LIN {X -0.037,Y -557.500,Z 807.101,A 0.000,B 0.000,C 90.000,E1 54.116} C_DIS
LIN {X -0.116,Y -555.159,Z 807.096,A 0.000,B 0.000,C 90.000,E1 53.290} C_DIS
LIN {X 0.105,Y -552.482,Z 807.091,A 0.000,B 0.000,C 90.000,E1 52.431} C_DIS
LIN {X -0.199,Y -550.629,Z 807.088,A 0.000,B 0.000,C 90.000,E1 51.904} C_DIS
LIN {X -0.029,Y -547.445,Z 807.084,A 0.000,B 0.000,C 90.000,E1 51.045} C_DIS
LIN {X -0.014,Y -545.178,Z 807.081,A 0.000,B 0.000,C 90.000,E1 50.481} C_DIS
LIN {X 0.251,Y -542.163,Z 807.077,A 0.000,B 0.000,C 90.000,E1 49.747} C_DIS
LIN {X -0.102,Y -537.935,Z 807.072,A 0.000,B 0.000,C 90.000,E1 48.933} C_DIS
LIN {X 0.083,Y -535.749,Z 807.069,A 0.000,B 0.000,C 90.000,E1 48.485} C_DIS
LIN {X -0.157,Y -531.502,Z 807.065,A 0.000,B 0.000,C 90.000,E1 47.796} C_DIS
LIN {X -0.128,Y -527.918,Z 807.062,A 0.000,B 0.000,C 90.000,E1 47.229} C_DIS
LIN {X 0.151,Y -523.761,Z 807.059,A 0.000,B 0.000,C 90.000,E1 46.620} C_DIS
LIN {X 0.098,Y -519.337,Z 807.056,A 0.000,B 0.000,C 90.000,E1 46.053} C_DIS
LIN {X 0.255,Y -514.772,Z 807.053,A 0.000,B 0.000,C 90.000,E1 45.486} C_DIS
LIN {X -0.036,Y -509.682,Z 807.050,A 0.000,B 0.000,C 90.000,E1 44.960} C_DIS
LIN {X 0.108,Y -505.640,Z 807.047,A 0.000,B 0.000,C 90.000,E1 44.514} C_DIS
LIN {X 0.235,Y -499.901,Z 807.044,A 0.000,B 0.000,C 90.000,E1 43.947} C_DIS
LIN {X -0.053,Y -495.627,Z 807.042,A 0.000,B 0.000,C 90.000,E1 43.581} C_DIS
LIN {X 0.080,Y -491.199,Z 807.040,A 0.000,B 0.000,C 90.000,E1 43.176} C_DIS
LIN {X -0.089,Y -484.986,Z 807.037,A 0.000,B 0.000,C 90.000,E1 42.690} C_DIS
LIN {X -0.041,Y -478.670,Z 807.034,A 0.000,B 0.000,C 90.000,E1 42.204} C_DIS
LIN {X 0.235,Y -470.752,Z 807.031,A 0.000,B 0.000,C 90.000,E1 41.595} C_DIS
LIN {X 0.146,Y -458.002,Z 807.026,A 0.000,B 0.000,C 90.000,E1 40.701} C_DIS
LIN {X -0.258,Y -443.553,Z 807.021,A 0.000,B 0.000,C 90.000,E1 39.725} C_DIS
LIN {X 0.027,Y -425.013,Z 807.013,A 0.000,B 0.000,C 90.000,E1 38.302} C_DIS
LIN {X 0.066,Y -412.541,Z 807.007,A 0.000,B 0.000,C 90.000,E1 37.282} C_DIS
LIN {X 0.050,Y -406.587,Z 807.004,A 0.000,B 0.000,C 90.000,E1 36.744} C_DIS
LIN {X -0.054,Y -402.832,Z 807.002,A 0.000,B 0.000,C 90.000,E1 36.377} C_DIS
LIN {X -0.143,Y -400.931,Z 807.001,A 0.000,B 0.000,C 90.000,E1 36.171} C_DIS
LIN {X 0.068,Y -400.912,Z 807.001,A 0.000,B 0.000,C 90.000,E1 36.137} C_DIS
LIN {X 0.061,Y -393.935,Z 806.977,A 0.000,B 0.000,C 90.000,E1 31.926} C_DIS
LIN {X 0.057,Y -393.844,Z 806.977,A 0.000,B 0.000,C 90.000,E1 31.750} C_DIS
LIN {X 0.223,Y -394.432,Z 806.968,A 0.000,B 0.000,C 90.000,E1 30.129} C_DIS
LIN {X -0.005,Y -395.827,Z 806.952,A 0.000,B 0.000,C 90.000,E1 27.334} C_DIS
LIN {X 0.124,Y -397.370,Z 806.938,A 0.000,B 0.000,C 90.000,E1 24.847} C_DIS
LIN {X 0.194,Y -398.558,Z 806.928,A 0.000,B 0.000,C 90.000,E1 23.078} C_DIS
LIN {X 0.069,Y -401.201,Z 806.911,A 0.000,B 0.000,C 90.000,E1 19.939} C_DIS
LIN {X 0.024,Y -404.592,Z 806.893,A 0.000,B 0.000,C 90.000,E1 16.804} C_DIS
LIN {X -0.103,Y -410.004,Z 806.872,A 0.000,B 0.000,C 90.000,E1 13.008} C_DIS
LIN {X -0.164,Y -413.482,Z 806.861,A 0.000,B 0.000,C 90.000,E1 10.950} C_DIS
LIN {X 0.106,Y -417.010,Z 806.849,A 0.000,B 0.000,C 90.000,E1 8.859} C_DIS
LIN {X -0.011,Y -420.720,Z 806.838,A 0.000,B 0.000,C 90.000,E1 6.834} C_DIS
LIN {X -0.173,Y -423.819,Z 806.829,A 0.000,B 0.000,C 90.000,E1 5.163} C_DIS
LIN {X -0.111,Y -428.905,Z 806.814,A 0.000,B 0.000,C 90.000,E1 2.465} C_DIS
LIN {X -0.089,Y -432.974,Z 806.803,A 0.000,B 0.000,C 90.000,E1 0.458} C_DIS
LIN {X 0.106,Y -437.263,Z 806.792,A 0.000,B 0.000,C 90.000,E1 358.453} C_DIS
LIN {X 0.025,Y -442.582,Z 806.779,A 0.000,B 0.000,C 90.000,E1 356.159} C_DIS
LIN {X -0.014,Y -447.421,Z 806.768,A 0.000,B 0.000,C 90.000,E1 354.204} C_DIS
LIN {X 0.034,Y -449.816,Z 806.762,A 0.000,B 0.000,C 90.000,E1 353.223} C_DIS
LIN {X -0.171,Y -454.610,Z 806.752,A 0.000,B 0.000,C 90.000,E1 351.310} C_DIS
LIN {X 0.180,Y -458.005,Z 806.745,A 0.000,B 0.000,C 90.000,E1 349.982} C_DIS
LIN {X -0.105,Y -461.068,Z 806.740,A 0.000,B 0.000,C 90.000,E1 349.218} C_DIS
LIN {X -0.029,Y -461.819,Z 806.739,A 0.000,B 0.000,C 90.000,E1 349.050} C_DIS
LIN {X -0.071,Y -464.733,Z 806.737,A 0.000,B 0.000,C 90.000,E1 348.578} C_DIS
LIN {X -0.200,Y -469.773,Z 806.734,A 0.000,B 0.000,C 90.000,E1 348.049} C_DIS
LIN {X -0.183,Y -473.009,Z 806.732,A 0.000,B 0.000,C 90.000,E1 347.757} C_DIS
LIN {X -0.111,Y -477.733,Z 806.730,A 0.000,B 0.000,C 90.000,E1 347.353} C_DIS
LIN {X 0.184,Y -498.420,Z 806.722,A 0.000,B 0.000,C 90.000,E1 345.880} C_DIS
LIN {X -0.191,Y -515.872,Z 806.715,A 0.000,B 0.000,C 90.000,E1 344.755} C_DIS
LIN {X 0.127,Y -528.321,Z 806.711,A 0.000,B 0.000,C 90.000,E1 343.866} C_DIS
LIN {X -0.178,Y -537.489,Z 806.707,A 0.000,B 0.000,C 90.000,E1 343.251} C_DIS
LIN {X 0.096,Y -544.938,Z 806.704,A 0.000,B 0.000,C 90.000,E1 342.670} C_DIS
LIN {X -0.147,Y -553.624,Z 806.700,A 0.000,B 0.000,C 90.000,E1 342.000} C_DIS
LIN {X -0.050,Y -557.840,Z 806.698,A 0.000,B 0.000,C 90.000,E1 341.638} C_DIS
LIN {X -0.131,Y -563.251,Z 806.695,A 0.000,B 0.000,C 90.000,E1 341.148} C_DIS
LIN {X 0.178,Y -568.543,Z 806.692,A 0.000,B 0.000,C 90.000,E1 340.604} C_DIS
LIN {X -0.137,Y -572.364,Z 806.690,A 0.000,B 0.000,C 90.000,E1 340.242} C_DIS
LIN {X -0.189,Y -578.188,Z 806.686,A 0.000,B 0.000,C 90.000,E1 339.571} C_DIS
LIN {X 0.115,Y -581.525,Z 806.684,A 0.000,B 0.000,C 90.000,E1 339.135} C_DIS
LIN {X 0.028,Y -587.428,Z 806.680,A 0.000,B 0.000,C 90.000,E1 338.337} C_DIS
LIN {X 0.110,Y -591.139,Z 806.677,A 0.000,B 0.000,C 90.000,E1 337.794} C_DIS
LIN {X 0.111,Y -596.462,Z 806.672,A 0.000,B 0.000,C 90.000,E1 336.997} C_DIS
LIN {X -0.149,Y -601.425,Z 806.668,A 0.000,B 0.000,C 90.000,E1 336.230} C_DIS
LIN {X -0.107,Y -607.823,Z 806.662,A 0.000,B 0.000,C 90.000,E1 335.177} C_DIS
LIN {X -0.265,Y -613.183,Z 806.657,A 0.000,B 0.000,C 90.000,E1 334.280} C_DIS
LIN {X 0.183,Y -619.697,Z 806.651,A 0.000,B 0.000,C 90.000,E1 333.076} C_DIS
LIN {X -0.384,Y -625.175,Z 806.645,A 0.000,B 0.000,C 90.000,E1 332.103} C_DIS
LIN {X -0.041,Y -629.543,Z 806.640,A 0.000,B 0.000,C 90.000,E1 331.179} C_DIS
LIN {X 0.381,Y -634.362,Z 806.634,A 0.000,B 0.000,C 90.000,E1 330.127} C_DIS
LIN {X -0.011,Y -639.079,Z 806.629,A 0.000,B 0.000,C 90.000,E1 329.154} C_DIS
LIN {X -0.081,Y -642.409,Z 806.625,A 0.000,B 0.000,C 90.000,E1 328.408} C_DIS
LIN {X -0.116,Y -645.450,Z 806.620,A 0.000,B 0.000,C 90.000,E1 327.661} C_DIS
LIN {X -0.167,Y -650.317,Z 806.613,A 0.000,B 0.000,C 90.000,E1 326.421} C_DIS
LIN {X -0.125,Y -653.040,Z 806.609,A 0.000,B 0.000,C 90.000,E1 325.674} C_DIS
LIN {X -0.141,Y -656.385,Z 806.604,A 0.000,B 0.000,C 90.000,E1 324.689} C_DIS
LIN {X -0.112,Y -659.436,Z 806.598,A 0.000,B 0.000,C 90.000,E1 323.703} C_DIS
LIN {X -0.132,Y -661.689,Z 806.594,A 0.000,B 0.000,C 90.000,E1 322.970} C_DIS
LIN {X -0.067,Y -665.082,Z 806.587,A 0.000,B 0.000,C 90.000,E1 321.743} C_DIS
LIN {X 0.043,Y -668.206,Z 806.581,A 0.000,B 0.000,C 90.000,E1 320.517} C_DIS
LIN {X 0.111,Y -670.998,Z 806.574,A 0.000,B 0.000,C 90.000,E1 319.299} C_DIS
LIN {X 0.214,Y -673.109,Z 806.569,A 0.000,B 0.000,C 90.000,E1 318.324} C_DIS
LIN {X -0.161,Y -675.018,Z 806.563,A 0.000,B 0.000,C 90.000,E1 317.391} C_DIS
LIN {X -0.450,Y -677.649,Z 806.555,A 0.000,B 0.000,C 90.000,E1 315.972} C_DIS
LIN {X -0.416,Y -678.098,Z 806.554,A 0.000,B 0.000,C 90.000,E1 315.729} C_DIS
LIN {X -0.174,Y -680.133,Z 806.546,A 0.000,B 0.000,C 90.000,E1 314.271} C_DIS
LIN {X 0.005,Y -681.446,Z 806.541,A 0.000,B 0.000,C 90.000,E1 313.299} C_DIS
LIN {X 0.284,Y -682.974,Z 806.534,A 0.000,B 0.000,C 90.000,E1 312.081} C_DIS
LIN {X 0.081,Y -684.417,Z 806.527,A 0.000,B 0.000,C 90.000,E1 310.906} C_DIS
LIN {X 0.018,Y -685.924,Z 806.519,A 0.000,B 0.000,C 90.000,E1 309.483} C_DIS
LIN {X -0.072,Y -687.086,Z 806.513,A 0.000,B 0.000,C 90.000,E1 308.302} C_DIS
LIN {X 0.024,Y -688.401,Z 806.505,A 0.000,B 0.000,C 90.000,E1 306.870} C_DIS
LIN {X 0.147,Y -689.583,Z 806.497,A 0.000,B 0.000,C 90.000,E1 305.438} C_DIS
LIN {X -0.142,Y -690.502,Z 806.490,A 0.000,B 0.000,C 90.000,E1 304.278} C_DIS
LIN {X -0.163,Y -691.695,Z 806.481,A 0.000,B 0.000,C 90.000,E1 302.625} C_DIS
LIN {X 0.056,Y -693.170,Z 806.471,A 0.000,B 0.000,C 90.000,E1 300.718} C_DIS
LIN {X -0.296,Y -694.103,Z 806.463,A 0.000,B 0.000,C 90.000,E1 299.333} C_DIS
LIN {X 0.228,Y -695.151,Z 806.454,A 0.000,B 0.000,C 90.000,E1 297.641} C_DIS
LIN {X -0.215,Y -696.425,Z 806.443,A 0.000,B 0.000,C 90.000,E1 295.796} C_DIS
LIN {X -0.104,Y -697.186,Z 806.438,A 0.000,B 0.000,C 90.000,E1 294.847} C_DIS
LIN {X -0.219,Y -697.383,Z 806.435,A 0.000,B 0.000,C 90.000,E1 294.387} C_DIS
LIN {X 0.039,Y -697.356,Z 806.434,A 0.000,B 0.000,C 90.000,E1 294.131} C_DIS
LIN {X 0.273,Y -696.938,Z 806.432,A 0.000,B 0.000,C 90.000,E1 293.643} C_DIS
LIN {X -0.110,Y -696.321,Z 806.430,A 0.000,B 0.000,C 90.000,E1 293.439} C_DIS
LIN {X 0.121,Y -694.445,Z 806.428,A 0.000,B 0.000,C 90.000,E1 292.950} C_DIS
LIN {X 0.245,Y -693.752,Z 806.427,A 0.000,B 0.000,C 90.000,E1 292.823} C_DIS
LIN {X 0.100,Y -692.715,Z 806.426,A 0.000,B 0.000,C 90.000,E1 292.717} C_DIS
LIN {X 0.220,Y -691.283,Z 806.426,A 0.000,B 0.000,C 90.000,E1 292.589} C_DIS
LIN {X 0.129,Y -686.698,Z 806.424,A 0.000,B 0.000,C 90.000,E1 292.280} C_DIS
LIN {X -0.136,Y -685.084,Z 806.423,A 0.000,B 0.000,C 90.000,E1 292.206} C_DIS
LIN {X 0.232,Y -682.669,Z 806.423,A 0.000,B 0.000,C 90.000,E1 292.078} C_DIS
LIN {X 0.207,Y -675.226,Z 806.422,A 0.000,B 0.000,C 90.000,E1 291.844} C_DIS
LIN {X 0.189,Y -673.325,Z 806.421,A 0.000,B 0.000,C 90.000,E1 291.791} C_DIS
LIN {X -0.184,Y -664.792,Z 806.420,A 0.000,B 0.000,C 90.000,E1 291.663} C_DIS
LIN {X -0.168,Y -648.502,Z 806.419,A 0.000,B 0.000,C 90.000,E1 291.408} C_DIS
LIN {X 0.368,Y -627.611,Z 806.417,A 0.000,B 0.000,C 90.000,E1 290.972} C_DIS
LIN {X -0.380,Y -614.207,Z 806.415,A 0.000,B 0.000,C 90.000,E1 290.737} C_DIS
LIN {X 0.116,Y -604.662,Z 806.414,A 0.000,B 0.000,C 90.000,E1 290.429} C_DIS
LIN {X -0.075,Y -595.597,Z 806.412,A 0.000,B 0.000,C 90.000,E1 290.120} C_DIS
LIN {X -0.078,Y -590.879,Z 806.411,A 0.000,B 0.000,C 90.000,E1 289.939} C_DIS
LIN {X -0.260,Y -587.841,Z 806.410,A 0.000,B 0.000,C 90.000,E1 289.812} C_DIS
LIN {X 0.019,Y -585.447,Z 806.409,A 0.000,B 0.000,C 90.000,E1 289.631} C_DIS
LIN {X -0.206,Y -582.531,Z 806.408,A 0.000,B 0.000,C 90.000,E1 289.504} C_DIS
LIN {X 0.311,Y -582.496,Z 806.408,A 0.000,B 0.000,C 90.000,E1 289.450} C_DIS
LIN {X 0.310,Y -581.681,Z 806.407,A 0.000,B 0.000,C 90.000,E1 289.268} C_DIS
LIN {X -0.111,Y -582.551,Z 806.405,A 0.000,B 0.000,C 90.000,E1 288.906} C_DIS
LIN {X 0.284,Y -583.583,Z 806.404,A 0.000,B 0.000,C 90.000,E1 288.598} C_DIS
LIN {X 0.140,Y -587.254,Z 806.400,A 0.000,B 0.000,C 90.000,E1 287.946} C_DIS
LIN {X 0.160,Y -591.295,Z 806.396,A 0.000,B 0.000,C 90.000,E1 287.275} C_DIS
LIN {X -0.028,Y -595.685,Z 806.392,A 0.000,B 0.000,C 90.000,E1 286.496} C_DIS
LIN {X 0.245,Y -596.903,Z 806.390,A 0.000,B 0.000,C 90.000,E1 286.205} C_DIS
LIN {X 0.109,Y -600.031,Z 806.386,A 0.000,B 0.000,C 90.000,E1 285.426} C_DIS
LIN {X -0.178,Y -600.898,Z 806.384,A 0.000,B 0.000,C 90.000,E1 285.190} C_DIS
LIN {X -0.006,Y -602.048,Z 806.381,A 0.000,B 0.000,C 90.000,E1 284.647} C_DIS
LIN {X 0.022,Y -602.938,Z 806.378,A 0.000,B 0.000,C 90.000,E1 284.120} C_DIS
LIN {X -0.254,Y -603.285,Z 806.377,A 0.000,B 0.000,C 90.000,E1 283.883} C_DIS
LIN {X -0.214,Y -603.288,Z 806.374,A 0.000,B 0.000,C 90.000,E1 283.355} C_DIS
LIN {X -0.171,Y -602.957,Z 806.371,A 0.000,B 0.000,C 90.000,E1 282.827} C_DIS
LIN {X 0.144,Y -602.625,Z 806.370,A 0.000,B 0.000,C 90.000,E1 282.535} C_DIS
LIN {X 0.184,Y -601.388,Z 806.367,A 0.000,B 0.000,C 90.000,E1 282.007} C_DIS
LIN {X 0.215,Y -599.980,Z 806.364,A 0.000,B 0.000,C 90.000,E1 281.478} C_DIS
LIN {X 0.235,Y -597.951,Z 806.361,A 0.000,B 0.000,C 90.000,E1 280.950} C_DIS
LIN {X -0.256,Y -596.181,Z 806.359,A 0.000,B 0.000,C 90.000,E1 280.602} C_DIS
LIN {X 0.035,Y -594.900,Z 806.357,A 0.000,B 0.000,C 90.000,E1 280.310} C_DIS
LIN {X -0.088,Y -591.719,Z 806.354,A 0.000,B 0.000,C 90.000,E1 279.792} C_DIS
LIN {X 0.077,Y -588.827,Z 806.352,A 0.000,B 0.000,C 90.000,E1 279.378} C_DIS
LIN {X 0.242,Y -586.579,Z 806.351,A 0.000,B 0.000,C 90.000,E1 279.095} C_DIS
LIN {X 0.126,Y -585.159,Z 806.350,A 0.000,B 0.000,C 90.000,E1 278.973} C_DIS
LIN {X -0.083,Y -583.486,Z 806.349,A 0.000,B 0.000,C 90.000,E1 278.859} C_DIS
LIN {X -0.093,Y -581.758,Z 806.349,A 0.000,B 0.000,C 90.000,E1 278.746} C_DIS
LIN {X 0.246,Y -577.851,Z 806.347,A 0.000,B 0.000,C 90.000,E1 278.511} C_DIS
LIN {X -0.045,Y -569.845,Z 806.346,A 0.000,B 0.000,C 90.000,E1 278.276} C_DIS
LIN {X 0.054,Y -559.795,Z 806.345,A 0.000,B 0.000,C 90.000,E1 278.049} C_DIS
LIN {X 0.236,Y -556.972,Z 806.345,A 0.000,B 0.000,C 90.000,E1 277.992} C_DIS
LIN {X -0.197,Y -553.699,Z 806.344,A 0.000,B 0.000,C 90.000,E1 277.936} C_DIS
LIN {X 0.061,Y -553.337,Z 806.344,A 0.000,B 0.000,C 90.000,E1 277.871} C_DIS
LIN {X -0.192,Y -552.403,Z 806.343,A 0.000,B 0.000,C 90.000,E1 277.757} C_DIS
LIN {X -0.274,Y -551.492,Z 806.342,A 0.000,B 0.000,C 90.000,E1 277.644} C_DIS
LIN {X 0.188,Y -551.453,Z 806.342,A 0.000,B 0.000,C 90.000,E1 277.587} C_DIS
LIN {X 0.146,Y -551.448,Z 806.342,A 0.000,B 0.000,C 90.000,E1 277.587} C_DIS
LIN {X -0.026,Y -551.293,Z 806.341,A 0.000,B 0.000,C 90.000,E1 277.409} C_DIS
LIN {X -0.227,Y -550.912,Z 806.340,A 0.000,B 0.000,C 90.000,E1 277.239} C_DIS
LIN {X 0.166,Y -549.933,Z 806.332,A 0.000,B 0.000,C 90.000,E1 275.796} C_DIS
LIN {X -0.107,Y -549.514,Z 806.326,A 0.000,B 0.000,C 90.000,E1 274.702} C_DIS
LIN {X 0.119,Y -548.833,Z 806.320,A 0.000,B 0.000,C 90.000,E1 273.555} C_DIS
LIN {X -0.208,Y -548.137,Z 806.314,A 0.000,B 0.000,C 90.000,E1 272.465} C_DIS
LIN {X 0.135,Y -546.720,Z 806.303,A 0.000,B 0.000,C 90.000,E1 270.458} C_DIS
LIN {X -0.195,Y -545.795,Z 806.295,A 0.000,B 0.000,C 90.000,E1 269.083} C_DIS
LIN {X 0.144,Y -544.235,Z 806.282,A 0.000,B 0.000,C 90.000,E1 266.788} C_DIS
LIN {X -0.129,Y -543.053,Z 806.271,A 0.000,B 0.000,C 90.000,E1 264.837} C_DIS
LIN {X 0.119,Y -542.072,Z 806.263,A 0.000,B 0.000,C 90.000,E1 263.394} C_DIS
LIN {X -0.186,Y -540.898,Z 806.256,A 0.000,B 0.000,C 90.000,E1 262.008} C_DIS
LIN {X 0.082,Y -539.379,Z 806.246,A 0.000,B 0.000,C 90.000,E1 260.274} C_DIS
LIN {X -0.171,Y -538.251,Z 806.240,A 0.000,B 0.000,C 90.000,E1 259.162} C_DIS
LIN {X 0.158,Y -536.897,Z 806.232,A 0.000,B 0.000,C 90.000,E1 257.701} C_DIS
LIN {X 0.110,Y -535.129,Z 806.222,A 0.000,B 0.000,C 90.000,E1 255.992} C_DIS
LIN {X 0.201,Y -532.815,Z 806.211,A 0.000,B 0.000,C 90.000,E1 253.976} C_DIS
LIN {X -0.320,Y -530.792,Z 806.202,A 0.000,B 0.000,C 90.000,E1 252.308} C_DIS
LIN {X -0.240,Y -529.077,Z 806.194,A 0.000,B 0.000,C 90.000,E1 250.859} C_DIS
LIN {X -0.194,Y -527.535,Z 806.187,A 0.000,B 0.000,C 90.000,E1 249.699} C_DIS
LIN {X 0.002,Y -525.491,Z 806.179,A 0.000,B 0.000,C 90.000,E1 248.230} C_DIS
LIN {X -0.132,Y -523.365,Z 806.171,A 0.000,B 0.000,C 90.000,E1 246.794} C_DIS
LIN {X -0.300,Y -521.192,Z 806.163,A 0.000,B 0.000,C 90.000,E1 245.357} C_DIS
LIN {X 0.037,Y -519.355,Z 806.156,A 0.000,B 0.000,C 90.000,E1 244.152} C_DIS
LIN {X 0.027,Y -515.813,Z 806.145,A 0.000,B 0.000,C 90.000,E1 242.103} C_DIS
LIN {X -0.291,Y -513.076,Z 806.137,A 0.000,B 0.000,C 90.000,E1 240.667} C_DIS
LIN {X 0.035,Y -510.317,Z 806.129,A 0.000,B 0.000,C 90.000,E1 239.154} C_DIS
LIN {X -0.195,Y -507.992,Z 806.122,A 0.000,B 0.000,C 90.000,E1 237.995} C_DIS
LIN {X -0.135,Y -504.791,Z 806.114,A 0.000,B 0.000,C 90.000,E1 236.501} C_DIS
LIN {X -0.158,Y -502.316,Z 806.107,A 0.000,B 0.000,C 90.000,E1 235.308} C_DIS
LIN {X -0.213,Y -499.557,Z 806.101,A 0.000,B 0.000,C 90.000,E1 234.116} C_DIS
LIN {X 0.114,Y -495.036,Z 806.091,A 0.000,B 0.000,C 90.000,E1 232.271} C_DIS
LIN {X -0.002,Y -492.789,Z 806.085,A 0.000,B 0.000,C 90.000,E1 231.376} C_DIS
LIN {X 0.031,Y -485.624,Z 806.069,A 0.000,B 0.000,C 90.000,E1 228.324} C_DIS
LIN {X -0.212,Y -480.238,Z 806.055,A 0.000,B 0.000,C 90.000,E1 225.891} C_DIS
LIN {X -0.167,Y -476.113,Z 806.045,A 0.000,B 0.000,C 90.000,E1 224.028} C_DIS
LIN {X 0.026,Y -472.717,Z 806.036,A 0.000,B 0.000,C 90.000,E1 222.447} C_DIS
LIN {X 0.097,Y -467.428,Z 806.022,A 0.000,B 0.000,C 90.000,E1 219.930} C_DIS
LIN {X -0.144,Y -464.126,Z 806.013,A 0.000,B 0.000,C 90.000,E1 218.382} C_DIS
LIN {X -0.084,Y -460.861,Z 806.004,A 0.000,B 0.000,C 90.000,E1 216.790} C_DIS
LIN {X 0.220,Y -455.527,Z 805.990,A 0.000,B 0.000,C 90.000,E1 214.199} C_DIS
LIN {X -0.038,Y -452.264,Z 805.981,A 0.000,B 0.000,C 90.000,E1 212.625} C_DIS
LIN {X 0.106,Y -448.344,Z 805.971,A 0.000,B 0.000,C 90.000,E1 210.669} C_DIS
LIN {X -0.078,Y -444.464,Z 805.960,A 0.000,B 0.000,C 90.000,E1 208.743} C_DIS
LIN {X -0.224,Y -441.287,Z 805.951,A 0.000,B 0.000,C 90.000,E1 207.129} C_DIS
LIN {X -0.202,Y -437.595,Z 805.940,A 0.000,B 0.000,C 90.000,E1 205.155} C_DIS
LIN {X 0.121,Y -434.327,Z 805.930,A 0.000,B 0.000,C 90.000,E1 203.462} C_DIS
LIN {X -0.003,Y -429.806,Z 805.918,A 0.000,B 0.000,C 90.000,E1 201.153} C_DIS
LIN {X -0.114,Y -424.685,Z 805.903,A 0.000,B 0.000,C 90.000,E1 198.489} C_DIS
LIN {X 0.070,Y -420.794,Z 805.891,A 0.000,B 0.000,C 90.000,E1 196.441} C_DIS
LIN {X -0.126,Y -417.498,Z 805.882,A 0.000,B 0.000,C 90.000,E1 194.773} C_DIS
LIN {X -0.090,Y -414.261,Z 805.873,A 0.000,B 0.000,C 90.000,E1 193.063} C_DIS
LIN {X -0.093,Y -410.442,Z 805.861,A 0.000,B 0.000,C 90.000,E1 191.007} C_DIS
LIN {X 0.055,Y -406.743,Z 805.850,A 0.000,B 0.000,C 90.000,E1 188.916} C_DIS
LIN {X 0.052,Y -403.462,Z 805.840,A 0.000,B 0.000,C 90.000,E1 187.182} C_DIS
LIN {X -0.008,Y -400.980,Z 805.832,A 0.000,B 0.000,C 90.000,E1 185.796} C_DIS
LIN {X -0.177,Y -397.974,Z 805.823,A 0.000,B 0.000,C 90.000,E1 184.069} C_DIS
LIN {X -0.063,Y -392.546,Z 805.801,A 0.000,B 0.000,C 90.000,E1 180.172} C_DIS
LIN {X 0.175,Y -389.636,Z 805.787,A 0.000,B 0.000,C 90.000,E1 177.650} C_DIS
LIN {X -0.073,Y -388.507,Z 805.781,A 0.000,B 0.000,C 90.000,E1 176.617} C_DIS
LIN {X 0.081,Y -385.777,Z 805.767,A 0.000,B 0.000,C 90.000,E1 174.090} C_DIS
LIN {X -0.030,Y -383.509,Z 805.755,A 0.000,B 0.000,C 90.000,E1 171.951} C_DIS
LIN {X -0.048,Y -381.888,Z 805.745,A 0.000,B 0.000,C 90.000,E1 170.151} C_DIS
LIN {X 0.141,Y -379.406,Z 805.729,A 0.000,B 0.000,C 90.000,E1 167.229} C_DIS
LIN {X 0.054,Y -377.533,Z 805.715,A 0.000,B 0.000,C 90.000,E1 164.700} C_DIS
LIN {X -0.181,Y -375.922,Z 805.697,A 0.000,B 0.000,C 90.000,E1 161.456} C_DIS
LIN {X -0.183,Y -375.346,Z 805.683,A 0.000,B 0.000,C 90.000,E1 158.901} C_DIS
LIN {X -0.185,Y -375.706,Z 805.664,A 0.000,B 0.000,C 90.000,E1 155.613} C_DIS
LIN {X 0.074,Y -376.792,Z 805.652,A 0.000,B 0.000,C 90.000,E1 153.384} C_DIS
LIN {X 0.011,Y -379.478,Z 805.638,A 0.000,B 0.000,C 90.000,E1 150.845} C_DIS
LIN {X -0.087,Y -382.025,Z 805.630,A 0.000,B 0.000,C 90.000,E1 149.410} C_DIS
LIN {X 0.074,Y -383.792,Z 805.626,A 0.000,B 0.000,C 90.000,E1 148.663} C_DIS
LIN {X -0.099,Y -386.398,Z 805.621,A 0.000,B 0.000,C 90.000,E1 147.788} C_DIS
LIN {X -0.084,Y -388.278,Z 805.618,A 0.000,B 0.000,C 90.000,E1 147.248} C_DIS
LIN {X -0.097,Y -390.773,Z 805.614,A 0.000,B 0.000,C 90.000,E1 146.548} C_DIS
LIN {X 0.143,Y -393.979,Z 805.610,A 0.000,B 0.000,C 90.000,E1 145.801} C_DIS
LIN {X -0.041,Y -396.643,Z 805.607,A 0.000,B 0.000,C 90.000,E1 145.308} C_DIS
LIN {X -0.078,Y -400.780,Z 805.603,A 0.000,B 0.000,C 90.000,E1 144.609} C_DIS
LIN {X 0.020,Y -404.295,Z 805.600,A 0.000,B 0.000,C 90.000,E1 144.069} C_DIS
LIN {X -0.214,Y -413.312,Z 805.594,A 0.000,B 0.000,C 90.000,E1 142.924} C_DIS
LIN {X 0.000,Y -424.271,Z 805.587,A 0.000,B 0.000,C 90.000,E1 141.662} C_DIS
LIN {X 0.031,Y -429.654,Z 805.583,A 0.000,B 0.000,C 90.000,E1 141.009} C_DIS
LIN {X -0.130,Y -439.865,Z 805.576,A 0.000,B 0.000,C 90.000,E1 139.703} C_DIS
LIN {X 0.104,Y -446.170,Z 805.572,A 0.000,B 0.000,C 90.000,E1 138.852} C_DIS
LIN {X 0.152,Y -455.314,Z 805.565,A 0.000,B 0.000,C 90.000,E1 137.715} C_DIS
LIN {X 0.218,Y -460.035,Z 805.562,A 0.000,B 0.000,C 90.000,E1 137.067} C_DIS
LIN {X -0.014,Y -464.335,Z 805.558,A 0.000,B 0.000,C 90.000,E1 136.458} C_DIS
LIN {X -0.172,Y -477.324,Z 805.547,A 0.000,B 0.000,C 90.000,E1 134.433} C_DIS
LIN {X 0.176,Y -483.191,Z 805.542,A 0.000,B 0.000,C 90.000,E1 133.461} C_DIS
LIN {X 0.167,Y -491.525,Z 805.534,A 0.000,B 0.000,C 90.000,E1 132.081} C_DIS
LIN {X -0.196,Y -494.989,Z 805.531,A 0.000,B 0.000,C 90.000,E1 131.515} C_DIS
LIN {X -0.143,Y -504.022,Z 805.521,A 0.000,B 0.000,C 90.000,E1 129.850} C_DIS
LIN {X 0.058,Y -511.764,Z 805.513,A 0.000,B 0.000,C 90.000,E1 128.338} C_DIS
LIN {X 0.002,Y -518.944,Z 805.505,A 0.000,B 0.000,C 90.000,E1 126.870} C_DIS
LIN {X -0.208,Y -524.279,Z 805.498,A 0.000,B 0.000,C 90.000,E1 125.724} C_DIS
LIN {X 0.107,Y -527.837,Z 805.494,A 0.000,B 0.000,C 90.000,E1 124.818} C_DIS
LIN {X -0.134,Y -531.610,Z 805.488,A 0.000,B 0.000,C 90.000,E1 123.833} C_DIS
LIN {X 0.122,Y -534.492,Z 805.484,A 0.000,B 0.000,C 90.000,E1 123.086} C_DIS
LIN {X -0.025,Y -538.937,Z 805.478,A 0.000,B 0.000,C 90.000,E1 121.957} C_DIS
LIN {X -0.295,Y -542.012,Z 805.473,A 0.000,B 0.000,C 90.000,E1 121.131} C_DIS
LIN {X -0.074,Y -544.846,Z 805.468,A 0.000,B 0.000,C 90.000,E1 120.256} C_DIS
LIN {X -0.075,Y -548.311,Z 805.462,A 0.000,B 0.000,C 90.000,E1 119.127} C_DIS
LIN {X 0.191,Y -551.559,Z 805.456,A 0.000,B 0.000,C 90.000,E1 117.975} C_DIS
LIN {X 0.248,Y -553.701,Z 805.451,A 0.000,B 0.000,C 90.000,E1 117.129} C_DIS
LIN {X 0.076,Y -555.541,Z 805.446,A 0.000,B 0.000,C 90.000,E1 116.309} C_DIS
LIN {X 0.247,Y -557.849,Z 805.439,A 0.000,B 0.000,C 90.000,E1 114.899} C_DIS
LIN {X -0.089,Y -559.312,Z 805.432,A 0.000,B 0.000,C 90.000,E1 113.823} C_DIS
LIN {X 0.103,Y -560.602,Z 805.426,A 0.000,B 0.000,C 90.000,E1 112.695} C_DIS
LIN {X -0.113,Y -561.993,Z 805.419,A 0.000,B 0.000,C 90.000,E1 111.334} C_DIS
LIN {X 0.108,Y -562.648,Z 805.414,A 0.000,B 0.000,C 90.000,E1 110.482} C_DIS
LIN {X -0.061,Y -563.241,Z 805.408,A 0.000,B 0.000,C 90.000,E1 109.396} C_DIS
LIN {X -0.037,Y -563.706,Z 805.402,A 0.000,B 0.000,C 90.000,E1 108.290} C_DIS
LIN {X 0.028,Y -564.544,Z 805.389,A 0.000,B 0.000,C 90.000,E1 106.079} C_DIS
LIN {X -0.194,Y -565.506,Z 805.379,A 0.000,B 0.000,C 90.000,E1 104.175} C_DIS
LIN {X 0.063,Y -566.969,Z 805.366,A 0.000,B 0.000,C 90.000,E1 101.951} C_DIS
LIN {X 0.186,Y -568.338,Z 805.356,A 0.000,B 0.000,C 90.000,E1 100.018} C_DIS
LIN {X -0.135,Y -569.364,Z 805.348,A 0.000,B 0.000,C 90.000,E1 98.681} C_DIS
LIN {X 0.041,Y -570.288,Z 805.341,A 0.000,B 0.000,C 90.000,E1 97.296} C_DIS
LIN {X -0.059,Y -570.807,Z 805.336,A 0.000,B 0.000,C 90.000,E1 96.486} C_DIS
LIN {X 0.084,Y -571.578,Z 805.328,A 0.000,B 0.000,C 90.000,E1 95.106} C_DIS
LIN {X 0.244,Y -572.276,Z 805.321,A 0.000,B 0.000,C 90.000,E1 93.726} C_DIS
LIN {X -0.193,Y -572.877,Z 805.313,A 0.000,B 0.000,C 90.000,E1 92.407} C_DIS
LIN {X 0.238,Y -573.574,Z 805.303,A 0.000,B 0.000,C 90.000,E1 90.458} C_DIS
LIN {X -0.046,Y -574.120,Z 805.294,A 0.000,B 0.000,C 90.000,E1 88.854} C_DIS
LIN {X 0.121,Y -574.471,Z 805.286,A 0.000,B 0.000,C 90.000,E1 87.478} C_DIS
LIN {X -0.100,Y -574.846,Z 805.277,A 0.000,B 0.000,C 90.000,E1 85.869} C_DIS
LIN {X 0.123,Y -575.129,Z 805.270,A 0.000,B 0.000,C 90.000,E1 84.489} C_DIS
LIN {X -0.230,Y -575.430,Z 805.262,A 0.000,B 0.000,C 90.000,E1 83.166} C_DIS
LIN {X 0.012,Y -575.886,Z 805.250,A 0.000,B 0.000,C 90.000,E1 80.971} C_DIS
LIN {X 0.237,Y -576.269,Z 805.239,A 0.000,B 0.000,C 90.000,E1 79.050} C_DIS
LIN {X -0.048,Y -576.392,Z 805.233,A 0.000,B 0.000,C 90.000,E1 77.993} C_DIS
LIN {X -0.118,Y -576.462,Z 805.226,A 0.000,B 0.000,C 90.000,E1 76.645} C_DIS
LIN {X 0.296,Y -576.416,Z 805.220,A 0.000,B 0.000,C 90.000,E1 75.519} C_DIS
LIN {X 0.157,Y -576.335,Z 805.214,A 0.000,B 0.000,C 90.000,E1 74.448} C_DIS
LIN {X 0.028,Y -576.153,Z 805.205,A 0.000,B 0.000,C 90.000,E1 72.834} C_DIS
LIN {X 0.245,Y -575.914,Z 805.197,A 0.000,B 0.000,C 90.000,E1 71.456} C_DIS
LIN {X 0.098,Y -575.343,Z 805.187,A 0.000,B 0.000,C 90.000,E1 69.571} C_DIS
LIN {X -0.071,Y -574.833,Z 805.179,A 0.000,B 0.000,C 90.000,E1 68.230} C_DIS
LIN {X -0.042,Y -574.206,Z 805.172,A 0.000,B 0.000,C 90.000,E1 66.869} C_DIS
LIN {X 0.203,Y -573.509,Z 805.164,A 0.000,B 0.000,C 90.000,E1 65.485} C_DIS
LIN {X 0.079,Y -572.827,Z 805.158,A 0.000,B 0.000,C 90.000,E1 64.409} C_DIS
LIN {X 0.038,Y -571.903,Z 805.150,A 0.000,B 0.000,C 90.000,E1 63.050} C_DIS
LIN {X -0.114,Y -570.918,Z 805.144,A 0.000,B 0.000,C 90.000,E1 61.975} C_DIS
LIN {X -0.022,Y -569.723,Z 805.138,A 0.000,B 0.000,C 90.000,E1 60.873} C_DIS
LIN {X 0.015,Y -568.721,Z 805.134,A 0.000,B 0.000,C 90.000,E1 60.049} C_DIS
LIN {X 0.070,Y -567.182,Z 805.128,A 0.000,B 0.000,C 90.000,E1 58.948} C_DIS
LIN {X -0.098,Y -565.423,Z 805.121,A 0.000,B 0.000,C 90.000,E1 57.867} C_DIS
LIN {X 0.016,Y -563.361,Z 805.115,A 0.000,B 0.000,C 90.000,E1 56.755} C_DIS
LIN {X 0.011,Y -561.681,Z 805.111,A 0.000,B 0.000,C 90.000,E1 55.928} C_DIS
LIN {X 0.080,Y -559.052,Z 805.105,A 0.000,B 0.000,C 90.000,E1 54.815} C_DIS
LIN {X 0.022,Y -556.875,Z 805.100,A 0.000,B 0.000,C 90.000,E1 53.989} C_DIS
LIN {X 0.186,Y -555.340,Z 805.097,A 0.000,B 0.000,C 90.000,E1 53.417} C_DIS
LIN {X -0.028,Y -552.676,Z 805.092,A 0.000,B 0.000,C 90.000,E1 52.603} C_DIS
LIN {X 0.171,Y -549.737,Z 805.088,A 0.000,B 0.000,C 90.000,E1 51.743} C_DIS
LIN {X 0.282,Y -547.660,Z 805.084,A 0.000,B 0.000,C 90.000,E1 51.170} C_DIS
LIN {X 0.028,Y -542.876,Z 805.078,A 0.000,B 0.000,C 90.000,E1 50.070} C_DIS
LIN {X -0.168,Y -540.954,Z 805.076,A 0.000,B 0.000,C 90.000,E1 49.666} C_DIS
LIN {X 0.050,Y -537.382,Z 805.072,A 0.000,B 0.000,C 90.000,E1 48.933} C_DIS
LIN {X -0.171,Y -535.154,Z 805.070,A 0.000,B 0.000,C 90.000,E1 48.528} C_DIS
LIN {X -0.016,Y -530.818,Z 805.066,A 0.000,B 0.000,C 90.000,E1 47.796} C_DIS
LIN {X 0.002,Y -527.118,Z 805.062,A 0.000,B 0.000,C 90.000,E1 47.229} C_DIS
LIN {X -0.096,Y -522.899,Z 805.059,A 0.000,B 0.000,C 90.000,E1 46.662} C_DIS
LIN {X 0.033,Y -519.564,Z 805.057,A 0.000,B 0.000,C 90.000,E1 46.215} C_DIS
LIN {X 0.055,Y -514.861,Z 805.054,A 0.000,B 0.000,C 90.000,E1 45.648} C_DIS
LIN {X 0.108,Y -509.726,Z 805.051,A 0.000,B 0.000,C 90.000,E1 45.081} C_DIS
LIN {X -0.015,Y -505.735,Z 805.048,A 0.000,B 0.000,C 90.000,E1 44.676} C_DIS
LIN {X 0.233,Y -500.133,Z 805.045,A 0.000,B 0.000,C 90.000,E1 44.109} C_DIS
LIN {X -0.004,Y -493.097,Z 805.042,A 0.000,B 0.000,C 90.000,E1 43.500} C_DIS
LIN {X 0.132,Y -488.456,Z 805.040,A 0.000,B 0.000,C 90.000,E1 43.095} C_DIS
LIN {X 0.179,Y -482.401,Z 805.037,A 0.000,B 0.000,C 90.000,E1 42.609} C_DIS
LIN {X 0.029,Y -474.527,Z 805.034,A 0.000,B 0.000,C 90.000,E1 42.043} C_DIS
LIN {X 0.207,Y -463.356,Z 805.029,A 0.000,B 0.000,C 90.000,E1 41.229} C_DIS
LIN {X -0.012,Y -445.813,Z 805.022,A 0.000,B 0.000,C 90.000,E1 40.011} C_DIS
LIN {X -0.133,Y -426.715,Z 805.015,A 0.000,B 0.000,C 90.000,E1 38.624} C_DIS
LIN {X -0.183,Y -411.107,Z 805.008,A 0.000,B 0.000,C 90.000,E1 37.363} C_DIS
LIN {X -0.135,Y -406.610,Z 805.005,A 0.000,B 0.000,C 90.000,E1 36.950} C_DIS
LIN {X -0.009,Y -401.370,Z 805.002,A 0.000,B 0.000,C 90.000,E1 36.377} C_DIS
LIN {X -0.042,Y -401.353,Z 805.002,A 0.000,B 0.000,C 90.000,E1 36.377} C_DIS
LIN {X -0.047,Y -394.198,Z 804.979,A 0.000,B 0.000,C 90.000,E1 32.133} C_DIS
LIN {X 0.157,Y -394.028,Z 804.978,A 0.000,B 0.000,C 90.000,E1 31.926} C_DIS
LIN {X 0.155,Y -394.612,Z 804.969,A 0.000,B 0.000,C 90.000,E1 30.335} C_DIS
LIN {X -0.095,Y -395.791,Z 804.955,A 0.000,B 0.000,C 90.000,E1 27.897} C_DIS
LIN {X 0.023,Y -397.253,Z 804.941,A 0.000,B 0.000,C 90.000,E1 25.412} C_DIS
LIN {X 0.091,Y -398.440,Z 804.931,A 0.000,B 0.000,C 90.000,E1 23.643} C_DIS
LIN {X 0.192,Y -401.262,Z 804.912,A 0.000,B 0.000,C 90.000,E1 20.120} C_DIS
LIN {X 0.149,Y -404.622,Z 804.895,A 0.000,B 0.000,C 90.000,E1 16.985} C_DIS
LIN {X 0.010,Y -409.449,Z 804.875,A 0.000,B 0.000,C 90.000,E1 13.536} C_DIS
LIN {X -0.026,Y -413.396,Z 804.862,A 0.000,B 0.000,C 90.000,E1 11.130} C_DIS
LIN {X -0.161,Y -416.959,Z 804.850,A 0.000,B 0.000,C 90.000,E1 9.095} C_DIS
LIN {X 0.142,Y -420.641,Z 804.839,A 0.000,B 0.000,C 90.000,E1 7.011} C_DIS
LIN {X 0.027,Y -423.765,Z 804.830,A 0.000,B 0.000,C 90.000,E1 5.334} C_DIS
LIN {X 0.149,Y -429.463,Z 804.813,A 0.000,B 0.000,C 90.000,E1 2.293} C_DIS
LIN {X 0.165,Y -434.636,Z 804.799,A 0.000,B 0.000,C 90.000,E1 359.771} C_DIS
LIN {X 0.109,Y -440.484,Z 804.784,A 0.000,B 0.000,C 90.000,E1 357.135} C_DIS
LIN {X 0.149,Y -446.026,Z 804.771,A 0.000,B 0.000,C 90.000,E1 354.837} C_DIS
LIN {X 0.053,Y -450.039,Z 804.762,A 0.000,B 0.000,C 90.000,E1 353.223} C_DIS
LIN {X -0.147,Y -454.780,Z 804.752,A 0.000,B 0.000,C 90.000,E1 351.310} C_DIS
LIN {X 0.205,Y -458.138,Z 804.745,A 0.000,B 0.000,C 90.000,E1 349.982} C_DIS
LIN {X -0.061,Y -460.848,Z 804.740,A 0.000,B 0.000,C 90.000,E1 349.218} C_DIS
LIN {X -0.199,Y -463.187,Z 804.737,A 0.000,B 0.000,C 90.000,E1 348.757} C_DIS
LIN {X 0.089,Y -465.609,Z 804.735,A 0.000,B 0.000,C 90.000,E1 348.342} C_DIS
LIN {X 0.069,Y -469.780,Z 804.733,A 0.000,B 0.000,C 90.000,E1 347.881} C_DIS
LIN {X 0.205,Y -473.528,Z 804.731,A 0.000,B 0.000,C 90.000,E1 347.521} C_DIS
LIN {X -0.123,Y -479.550,Z 804.728,A 0.000,B 0.000,C 90.000,E1 347.061} C_DIS
LIN {X -0.198,Y -503.485,Z 804.719,A 0.000,B 0.000,C 90.000,E1 345.408} C_DIS
LIN {X -0.146,Y -517.729,Z 804.714,A 0.000,B 0.000,C 90.000,E1 344.448} C_DIS
LIN {X 0.046,Y -528.645,Z 804.709,A 0.000,B 0.000,C 90.000,E1 343.685} C_DIS
LIN {X 0.110,Y -537.759,Z 804.706,A 0.000,B 0.000,C 90.000,E1 343.032} C_DIS
LIN {X -0.038,Y -545.240,Z 804.703,A 0.000,B 0.000,C 90.000,E1 342.489} C_DIS
LIN {X 0.053,Y -553.721,Z 804.699,A 0.000,B 0.000,C 90.000,E1 341.819} C_DIS
LIN {X 0.176,Y -557.833,Z 804.697,A 0.000,B 0.000,C 90.000,E1 341.456} C_DIS
LIN {X -0.086,Y -566.001,Z 804.693,A 0.000,B 0.000,C 90.000,E1 340.732} C_DIS
LIN {X -0.248,Y -571.042,Z 804.690,A 0.000,B 0.000,C 90.000,E1 340.242} C_DIS
LIN {X -0.187,Y -575.844,Z 804.687,A 0.000,B 0.000,C 90.000,E1 339.699} C_DIS
LIN {X -0.264,Y -581.366,Z 804.683,A 0.000,B 0.000,C 90.000,E1 339.028} C_DIS
LIN {X -0.144,Y -587.315,Z 804.679,A 0.000,B 0.000,C 90.000,E1 338.209} C_DIS
LIN {X -0.123,Y -591.952,Z 804.675,A 0.000,B 0.000,C 90.000,E1 337.539} C_DIS
LIN {X 0.216,Y -595.505,Z 804.672,A 0.000,B 0.000,C 90.000,E1 336.975} C_DIS
LIN {X 0.152,Y -603.040,Z 804.666,A 0.000,B 0.000,C 90.000,E1 335.793} C_DIS
LIN {X -0.337,Y -609.387,Z 804.660,A 0.000,B 0.000,C 90.000,E1 334.793} C_DIS
LIN {X 0.092,Y -613.952,Z 804.656,A 0.000,B 0.000,C 90.000,E1 333.973} C_DIS
LIN {X -0.005,Y -620.410,Z 804.649,A 0.000,B 0.000,C 90.000,E1 332.820} C_DIS
LIN {X 0.280,Y -625.207,Z 804.644,A 0.000,B 0.000,C 90.000,E1 331.897} C_DIS
LIN {X -0.224,Y -629.563,Z 804.639,A 0.000,B 0.000,C 90.000,E1 331.051} C_DIS
LIN {X 0.231,Y -635.706,Z 804.632,A 0.000,B 0.000,C 90.000,E1 329.744} C_DIS
LIN {X 0.178,Y -640.331,Z 804.626,A 0.000,B 0.000,C 90.000,E1 328.742} C_DIS
LIN {X 0.125,Y -643.550,Z 804.622,A 0.000,B 0.000,C 90.000,E1 327.995} C_DIS
LIN {X 0.113,Y -649.529,Z 804.614,A 0.000,B 0.000,C 90.000,E1 326.501} C_DIS
LIN {X 0.148,Y -652.316,Z 804.610,A 0.000,B 0.000,C 90.000,E1 325.754} C_DIS
LIN {X 0.044,Y -656.580,Z 804.603,A 0.000,B 0.000,C 90.000,E1 324.529} C_DIS
LIN {X 0.163,Y -660.375,Z 804.596,A 0.000,B 0.000,C 90.000,E1 323.290} C_DIS
LIN {X -0.290,Y -663.288,Z 804.591,A 0.000,B 0.000,C 90.000,E1 322.351} C_DIS
LIN {X -0.271,Y -665.272,Z 804.587,A 0.000,B 0.000,C 90.000,E1 321.618} C_DIS
LIN {X -0.246,Y -667.856,Z 804.581,A 0.000,B 0.000,C 90.000,E1 320.642} C_DIS
LIN {X 0.333,Y -670.725,Z 804.575,A 0.000,B 0.000,C 90.000,E1 319.380} C_DIS
LIN {X 0.446,Y -673.390,Z 804.568,A 0.000,B 0.000,C 90.000,E1 318.162} C_DIS
LIN {X 0.053,Y -674.869,Z 804.564,A 0.000,B 0.000,C 90.000,E1 317.472} C_DIS
LIN {X -0.272,Y -677.095,Z 804.557,A 0.000,B 0.000,C 90.000,E1 316.296} C_DIS
LIN {X -0.168,Y -678.356,Z 804.553,A 0.000,B 0.000,C 90.000,E1 315.567} C_DIS
LIN {X 0.079,Y -680.439,Z 804.545,A 0.000,B 0.000,C 90.000,E1 314.109} C_DIS
LIN {X -0.206,Y -681.770,Z 804.540,A 0.000,B 0.000,C 90.000,E1 313.176} C_DIS
LIN {X 0.038,Y -683.309,Z 804.533,A 0.000,B 0.000,C 90.000,E1 311.962} C_DIS
LIN {X -0.101,Y -684.747,Z 804.527,A 0.000,B 0.000,C 90.000,E1 310.782} C_DIS
LIN {X 0.236,Y -686.023,Z 804.520,A 0.000,B 0.000,C 90.000,E1 309.564} C_DIS
LIN {X 0.150,Y -687.215,Z 804.513,A 0.000,B 0.000,C 90.000,E1 308.382} C_DIS
LIN {X 0.253,Y -688.535,Z 804.505,A 0.000,B 0.000,C 90.000,E1 306.950} C_DIS
LIN {X 0.382,Y -689.725,Z 804.498,A 0.000,B 0.000,C 90.000,E1 305.518} C_DIS
LIN {X 0.127,Y -690.820,Z 804.490,A 0.000,B 0.000,C 90.000,E1 304.119} C_DIS
LIN {X 0.087,Y -691.844,Z 804.482,A 0.000,B 0.000,C 90.000,E1 302.704} C_DIS
LIN {X 0.319,Y -693.298,Z 804.471,A 0.000,B 0.000,C 90.000,E1 300.797} C_DIS
LIN {X -0.024,Y -694.258,Z 804.463,A 0.000,B 0.000,C 90.000,E1 299.411} C_DIS
LIN {X -0.104,Y -695.285,Z 804.454,A 0.000,B 0.000,C 90.000,E1 297.769} C_DIS
LIN {X 0.386,Y -696.528,Z 804.444,A 0.000,B 0.000,C 90.000,E1 295.848} C_DIS
LIN {X -0.173,Y -697.400,Z 804.437,A 0.000,B 0.000,C 90.000,E1 294.719} C_DIS
LIN {X 0.349,Y -697.575,Z 804.435,A 0.000,B 0.000,C 90.000,E1 294.207} C_DIS
LIN {X -0.053,Y -697.156,Z 804.432,A 0.000,B 0.000,C 90.000,E1 293.770} C_DIS
LIN {X 0.205,Y -696.798,Z 804.431,A 0.000,B 0.000,C 90.000,E1 293.515} C_DIS
LIN {X -0.198,Y -694.929,Z 804.428,A 0.000,B 0.000,C 90.000,E1 293.078} C_DIS
LIN {X 0.050,Y -693.596,Z 804.427,A 0.000,B 0.000,C 90.000,E1 292.823} C_DIS
LIN {X -0.095,Y -692.497,Z 804.426,A 0.000,B 0.000,C 90.000,E1 292.717} C_DIS
LIN {X 0.146,Y -686.465,Z 804.424,A 0.000,B 0.000,C 90.000,E1 292.280} C_DIS
LIN {X -0.114,Y -684.760,Z 804.423,A 0.000,B 0.000,C 90.000,E1 292.206} C_DIS
LIN {X 0.121,Y -682.533,Z 804.423,A 0.000,B 0.000,C 90.000,E1 292.099} C_DIS
LIN {X 0.194,Y -674.346,Z 804.422,A 0.000,B 0.000,C 90.000,E1 291.844} C_DIS
LIN {X -0.411,Y -672.334,Z 804.421,A 0.000,B 0.000,C 90.000,E1 291.844} C_DIS
LIN {X -0.120,Y -663.454,Z 804.420,A 0.000,B 0.000,C 90.000,E1 291.663} C_DIS
LIN {X 0.241,Y -649.108,Z 804.419,A 0.000,B 0.000,C 90.000,E1 291.408} C_DIS
LIN {X 0.179,Y -631.712,Z 804.417,A 0.000,B 0.000,C 90.000,E1 291.099} C_DIS
LIN {X -0.164,Y -621.419,Z 804.416,A 0.000,B 0.000,C 90.000,E1 290.918} C_DIS
LIN {X 0.123,Y -609.873,Z 804.415,A 0.000,B 0.000,C 90.000,E1 290.610} C_DIS
LIN {X 0.173,Y -601.944,Z 804.413,A 0.000,B 0.000,C 90.000,E1 290.375} C_DIS
LIN {X 0.089,Y -589.485,Z 804.411,A 0.000,B 0.000,C 90.000,E1 289.939} C_DIS
LIN {X -0.117,Y -582.439,Z 804.409,A 0.000,B 0.000,C 90.000,E1 289.631} C_DIS
LIN {X -0.032,Y -579.354,Z 804.408,A 0.000,B 0.000,C 90.000,E1 289.450} C_DIS
LIN {X 0.180,Y -577.779,Z 804.407,A 0.000,B 0.000,C 90.000,E1 289.268} C_DIS
LIN {X 0.150,Y -577.779,Z 804.407,A 0.000,B 0.000,C 90.000,E1 289.268} C_DIS
LIN {X 0.154,Y -577.715,Z 804.406,A 0.000,B 0.000,C 90.000,E1 289.141} C_DIS
LIN {X -0.202,Y -577.232,Z 804.405,A 0.000,B 0.000,C 90.000,E1 288.906} C_DIS
LIN {X -0.027,Y -577.695,Z 804.404,A 0.000,B 0.000,C 90.000,E1 288.725} C_DIS
LIN {X 0.348,Y -578.691,Z 804.403,A 0.000,B 0.000,C 90.000,E1 288.417} C_DIS
LIN {X -0.007,Y -580.113,Z 804.401,A 0.000,B 0.000,C 90.000,E1 288.181} C_DIS
LIN {X 0.251,Y -585.710,Z 804.396,A 0.000,B 0.000,C 90.000,E1 287.221} C_DIS
LIN {X 0.084,Y -589.358,Z 804.392,A 0.000,B 0.000,C 90.000,E1 286.567} C_DIS
LIN {X 0.188,Y -592.038,Z 804.389,A 0.000,B 0.000,C 90.000,E1 286.024} C_DIS
LIN {X 0.304,Y -594.272,Z 804.386,A 0.000,B 0.000,C 90.000,E1 285.481} C_DIS
LIN {X 0.275,Y -595.973,Z 804.383,A 0.000,B 0.000,C 90.000,E1 284.954} C_DIS
LIN {X -0.021,Y -596.778,Z 804.382,A 0.000,B 0.000,C 90.000,E1 284.717} C_DIS
LIN {X -0.316,Y -597.321,Z 804.380,A 0.000,B 0.000,C 90.000,E1 284.481} C_DIS
LIN {X -0.172,Y -597.961,Z 804.377,A 0.000,B 0.000,C 90.000,E1 283.939} C_DIS
LIN {X -0.170,Y -598.047,Z 804.374,A 0.000,B 0.000,C 90.000,E1 283.411} C_DIS
LIN {X -0.166,Y -597.688,Z 804.372,A 0.000,B 0.000,C 90.000,E1 282.883} C_DIS
LIN {X 0.128,Y -597.237,Z 804.370,A 0.000,B 0.000,C 90.000,E1 282.591} C_DIS
LIN {X 0.130,Y -596.063,Z 804.367,A 0.000,B 0.000,C 90.000,E1 282.063} C_DIS
LIN {X 0.123,Y -594.605,Z 804.364,A 0.000,B 0.000,C 90.000,E1 281.535} C_DIS
LIN {X 0.105,Y -592.440,Z 804.361,A 0.000,B 0.000,C 90.000,E1 281.007} C_DIS
LIN {X -0.141,Y -589.109,Z 804.358,A 0.000,B 0.000,C 90.000,E1 280.366} C_DIS
LIN {X -0.092,Y -586.330,Z 804.355,A 0.000,B 0.000,C 90.000,E1 279.962} C_DIS
LIN {X 0.160,Y -584.154,Z 804.354,A 0.000,B 0.000,C 90.000,E1 279.670} C_DIS
LIN {X -0.054,Y -582.973,Z 804.353,A 0.000,B 0.000,C 90.000,E1 279.557} C_DIS
LIN {X -0.271,Y -580.142,Z 804.352,A 0.000,B 0.000,C 90.000,E1 279.321} C_DIS
LIN {X 0.203,Y -578.098,Z 804.351,A 0.000,B 0.000,C 90.000,E1 279.151} C_DIS
LIN {X -0.071,Y -567.617,Z 804.349,A 0.000,B 0.000,C 90.000,E1 278.803} C_DIS
LIN {X -0.027,Y -561.513,Z 804.348,A 0.000,B 0.000,C 90.000,E1 278.624} C_DIS
LIN {X 0.035,Y -558.959,Z 804.348,A 0.000,B 0.000,C 90.000,E1 278.568} C_DIS
LIN {X -0.132,Y -554.358,Z 804.347,A 0.000,B 0.000,C 90.000,E1 278.454} C_DIS
LIN {X -0.086,Y -553.595,Z 804.347,A 0.000,B 0.000,C 90.000,E1 278.398} C_DIS
LIN {X -0.039,Y -553.122,Z 804.346,A 0.000,B 0.000,C 90.000,E1 278.341} C_DIS
LIN {X -0.055,Y -551.715,Z 804.345,A 0.000,B 0.000,C 90.000,E1 278.106} C_DIS
LIN {X -0.096,Y -551.696,Z 804.345,A 0.000,B 0.000,C 90.000,E1 278.106} C_DIS
LIN {X 0.231,Y -551.111,Z 804.343,A 0.000,B 0.000,C 90.000,E1 277.757} C_DIS
LIN {X -0.024,Y -550.429,Z 804.337,A 0.000,B 0.000,C 90.000,E1 276.663} C_DIS
LIN {X -0.284,Y -549.880,Z 804.331,A 0.000,B 0.000,C 90.000,E1 275.568} C_DIS
LIN {X -0.052,Y -549.548,Z 804.326,A 0.000,B 0.000,C 90.000,E1 274.702} C_DIS
LIN {X -0.247,Y -548.519,Z 804.317,A 0.000,B 0.000,C 90.000,E1 273.037} C_DIS
LIN {X 0.009,Y -547.537,Z 804.309,A 0.000,B 0.000,C 90.000,E1 271.604} C_DIS
LIN {X -0.223,Y -546.225,Z 804.298,A 0.000,B 0.000,C 90.000,E1 269.656} C_DIS
LIN {X 0.036,Y -545.006,Z 804.289,A 0.000,B 0.000,C 90.000,E1 267.936} C_DIS
LIN {X -0.250,Y -543.751,Z 804.278,A 0.000,B 0.000,C 90.000,E1 265.988} C_DIS
LIN {X 0.001,Y -542.897,Z 804.270,A 0.000,B 0.000,C 90.000,E1 264.546} C_DIS
LIN {X 0.178,Y -542.106,Z 804.263,A 0.000,B 0.000,C 90.000,E1 263.394} C_DIS
LIN {X -0.126,Y -540.943,Z 804.256,A 0.000,B 0.000,C 90.000,E1 262.008} C_DIS
LIN {X 0.212,Y -539.193,Z 804.245,A 0.000,B 0.000,C 90.000,E1 259.982} C_DIS
LIN {X 0.156,Y -537.245,Z 804.233,A 0.000,B 0.000,C 90.000,E1 257.993} C_DIS
LIN {X -0.008,Y -535.495,Z 804.224,A 0.000,B 0.000,C 90.000,E1 256.297} C_DIS
LIN {X 0.039,Y -533.564,Z 804.214,A 0.000,B 0.000,C 90.000,E1 254.574} C_DIS
LIN {X 0.044,Y -531.552,Z 804.205,A 0.000,B 0.000,C 90.000,E1 252.851} C_DIS
LIN {X -0.183,Y -529.514,Z 804.195,A 0.000,B 0.000,C 90.000,E1 251.148} C_DIS
LIN {X -0.303,Y -528.005,Z 804.189,A 0.000,B 0.000,C 90.000,E1 250.007} C_DIS
LIN {X -0.084,Y -526.402,Z 804.182,A 0.000,B 0.000,C 90.000,E1 248.827} C_DIS
LIN {X -0.225,Y -523.887,Z 804.173,A 0.000,B 0.000,C 90.000,E1 247.102} C_DIS
LIN {X -0.228,Y -521.255,Z 804.163,A 0.000,B 0.000,C 90.000,E1 245.357} C_DIS
LIN {X 0.109,Y -519.421,Z 804.156,A 0.000,B 0.000,C 90.000,E1 244.152} C_DIS
LIN {X 0.101,Y -515.892,Z 804.145,A 0.000,B 0.000,C 90.000,E1 242.103} C_DIS
LIN {X 0.130,Y -513.737,Z 804.139,A 0.000,B 0.000,C 90.000,E1 240.923} C_DIS
LIN {X 0.032,Y -510.950,Z 804.130,A 0.000,B 0.000,C 90.000,E1 239.459} C_DIS
LIN {X -0.017,Y -508.645,Z 804.124,A 0.000,B 0.000,C 90.000,E1 238.280} C_DIS
LIN {X 0.049,Y -505.524,Z 804.116,A 0.000,B 0.000,C 90.000,E1 236.786} C_DIS
LIN {X -0.078,Y -502.375,Z 804.107,A 0.000,B 0.000,C 90.000,E1 235.308} C_DIS
LIN {X -0.134,Y -499.626,Z 804.101,A 0.000,B 0.000,C 90.000,E1 234.116} C_DIS
LIN {X 0.194,Y -495.103,Z 804.091,A 0.000,B 0.000,C 90.000,E1 232.271} C_DIS
LIN {X 0.079,Y -492.839,Z 804.086,A 0.000,B 0.000,C 90.000,E1 231.376} C_DIS
LIN {X 0.112,Y -485.672,Z 804.069,A 0.000,B 0.000,C 90.000,E1 228.324} C_DIS
LIN {X -0.129,Y -480.311,Z 804.055,A 0.000,B 0.000,C 90.000,E1 225.891} C_DIS
LIN {X -0.083,Y -476.186,Z 804.045,A 0.000,B 0.000,C 90.000,E1 224.028} C_DIS
LIN {X 0.110,Y -472.778,Z 804.036,A 0.000,B 0.000,C 90.000,E1 222.447} C_DIS
LIN {X 0.114,Y -468.145,Z 804.024,A 0.000,B 0.000,C 90.000,E1 220.253} C_DIS
LIN {X -0.059,Y -464.197,Z 804.013,A 0.000,B 0.000,C 90.000,E1 218.382} C_DIS
LIN {X 0.003,Y -460.890,Z 804.004,A 0.000,B 0.000,C 90.000,E1 216.790} C_DIS
LIN {X 0.249,Y -458.859,Z 803.999,A 0.000,B 0.000,C 90.000,E1 215.804} C_DIS
LIN {X 0.033,Y -454.950,Z 803.988,A 0.000,B 0.000,C 90.000,E1 213.913} C_DIS
LIN {X -0.146,Y -451.006,Z 803.978,A 0.000,B 0.000,C 90.000,E1 212.005} C_DIS
LIN {X -0.040,Y -447.115,Z 803.967,A 0.000,B 0.000,C 90.000,E1 210.050} C_DIS
LIN {X -0.140,Y -443.886,Z 803.958,A 0.000,B 0.000,C 90.000,E1 208.437} C_DIS
LIN {X -0.249,Y -440.157,Z 803.947,A 0.000,B 0.000,C 90.000,E1 206.488} C_DIS
LIN {X -0.090,Y -437.008,Z 803.938,A 0.000,B 0.000,C 90.000,E1 204.823} C_DIS
LIN {X 0.042,Y -433.766,Z 803.929,A 0.000,B 0.000,C 90.000,E1 203.153} C_DIS
LIN {X 0.092,Y -429.926,Z 803.918,A 0.000,B 0.000,C 90.000,E1 201.153} C_DIS
LIN {X -0.016,Y -424.802,Z 803.903,A 0.000,B 0.000,C 90.000,E1 198.489} C_DIS
LIN {X -0.008,Y -421.542,Z 803.893,A 0.000,B 0.000,C 90.000,E1 196.804} C_DIS
LIN {X 0.163,Y -418.949,Z 803.886,A 0.000,B 0.000,C 90.000,E1 195.426} C_DIS
LIN {X -0.032,Y -415.009,Z 803.875,A 0.000,B 0.000,C 90.000,E1 193.411} C_DIS
LIN {X -0.102,Y -411.183,Z 803.863,A 0.000,B 0.000,C 90.000,E1 191.366} C_DIS
LIN {X 0.142,Y -407.497,Z 803.852,A 0.000,B 0.000,C 90.000,E1 189.265} C_DIS
LIN {X 0.201,Y -404.968,Z 803.844,A 0.000,B 0.000,C 90.000,E1 187.871} C_DIS
LIN {X 0.102,Y -401.143,Z 803.832,A 0.000,B 0.000,C 90.000,E1 185.796} C_DIS
LIN {X -0.060,Y -394.519,Z 803.809,A 0.000,B 0.000,C 90.000,E1 181.604} C_DIS
LIN {X 0.143,Y -391.037,Z 803.793,A 0.000,B 0.000,C 90.000,E1 178.740} C_DIS
LIN {X 0.051,Y -388.711,Z 803.781,A 0.000,B 0.000,C 90.000,E1 176.617} C_DIS
LIN {X -0.173,Y -386.025,Z 803.767,A 0.000,B 0.000,C 90.000,E1 174.147} C_DIS
LIN {X 0.030,Y -383.436,Z 803.753,A 0.000,B 0.000,C 90.000,E1 171.602} C_DIS
LIN {X 0.173,Y -382.452,Z 803.747,A 0.000,B 0.000,C 90.000,E1 170.500} C_DIS
LIN {X 0.113,Y -380.537,Z 803.735,A 0.000,B 0.000,C 90.000,E1 168.342} C_DIS
LIN {X -0.023,Y -378.596,Z 803.721,A 0.000,B 0.000,C 90.000,E1 165.825} C_DIS
LIN {X 0.013,Y -376.489,Z 803.701,A 0.000,B 0.000,C 90.000,E1 162.181} C_DIS
LIN {X 0.011,Y -375.728,Z 803.685,A 0.000,B 0.000,C 90.000,E1 159.263} C_DIS
LIN {X 0.030,Y -375.830,Z 803.667,A 0.000,B 0.000,C 90.000,E1 155.973} C_DIS
LIN {X 0.059,Y -377.217,Z 803.650,A 0.000,B 0.000,C 90.000,E1 153.050} C_DIS
LIN {X 0.014,Y -379.908,Z 803.636,A 0.000,B 0.000,C 90.000,E1 150.511} C_DIS
LIN {X 0.109,Y -381.770,Z 803.630,A 0.000,B 0.000,C 90.000,E1 149.410} C_DIS
LIN {X 0.089,Y -384.216,Z 803.624,A 0.000,B 0.000,C 90.000,E1 148.329} C_DIS
LIN {X 0.064,Y -386.264,Z 803.620,A 0.000,B 0.000,C 90.000,E1 147.612} C_DIS
LIN {X -0.066,Y -388.556,Z 803.616,A 0.000,B 0.000,C 90.000,E1 146.914} C_DIS
LIN {X -0.173,Y -391.216,Z 803.612,A 0.000,B 0.000,C 90.000,E1 146.215} C_DIS
LIN {X -0.049,Y -394.045,Z 803.609,A 0.000,B 0.000,C 90.000,E1 145.548} C_DIS
LIN {X -0.101,Y -397.346,Z 803.605,A 0.000,B 0.000,C 90.000,E1 144.895} C_DIS
LIN {X -0.081,Y -402.541,Z 803.600,A 0.000,B 0.000,C 90.000,E1 144.036} C_DIS
LIN {X -0.020,Y -408.429,Z 803.596,A 0.000,B 0.000,C 90.000,E1 143.210} C_DIS
LIN {X -0.047,Y -420.207,Z 803.587,A 0.000,B 0.000,C 90.000,E1 141.743} C_DIS
LIN {X 0.056,Y -425.410,Z 803.584,A 0.000,B 0.000,C 90.000,E1 141.126} C_DIS
LIN {X -0.029,Y -430.699,Z 803.581,A 0.000,B 0.000,C 90.000,E1 140.481} C_DIS
LIN {X 0.107,Y -439.678,Z 803.574,A 0.000,B 0.000,C 90.000,E1 139.299} C_DIS
LIN {X -0.258,Y -454.969,Z 803.563,A 0.000,B 0.000,C 90.000,E1 137.391} C_DIS
LIN {X 0.120,Y -459.773,Z 803.560,A 0.000,B 0.000,C 90.000,E1 136.701} C_DIS
LIN {X 0.232,Y -465.270,Z 803.555,A 0.000,B 0.000,C 90.000,E1 135.891} C_DIS
LIN {X -0.046,Y -475.432,Z 803.546,A 0.000,B 0.000,C 90.000,E1 134.352} C_DIS
LIN {X 0.077,Y -483.594,Z 803.539,A 0.000,B 0.000,C 90.000,E1 133.095} C_DIS
LIN {X 0.095,Y -488.489,Z 803.535,A 0.000,B 0.000,C 90.000,E1 132.324} C_DIS
LIN {X -0.287,Y -492.119,Z 803.532,A 0.000,B 0.000,C 90.000,E1 131.757} C_DIS
LIN {X -0.280,Y -495.511,Z 803.528,A 0.000,B 0.000,C 90.000,E1 131.148} C_DIS
LIN {X -0.246,Y -498.995,Z 803.525,A 0.000,B 0.000,C 90.000,E1 130.539} C_DIS
LIN {X -0.088,Y -503.196,Z 803.521,A 0.000,B 0.000,C 90.000,E1 129.769} C_DIS
LIN {X 0.189,Y -511.119,Z 803.513,A 0.000,B 0.000,C 90.000,E1 128.257} C_DIS
LIN {X -0.003,Y -517.745,Z 803.505,A 0.000,B 0.000,C 90.000,E1 126.950} C_DIS
LIN {X -0.273,Y -524.507,Z 803.497,A 0.000,B 0.000,C 90.000,E1 125.518} C_DIS
LIN {X 0.048,Y -528.171,Z 803.492,A 0.000,B 0.000,C 90.000,E1 124.612} C_DIS
LIN {X 0.082,Y -533.970,Z 803.484,A 0.000,B 0.000,C 90.000,E1 123.166} C_DIS
LIN {X 0.216,Y -538.435,Z 803.478,A 0.000,B 0.000,C 90.000,E1 122.005} C_DIS
LIN {X 0.130,Y -542.529,Z 803.472,A 0.000,B 0.000,C 90.000,E1 120.875} C_DIS
LIN {X -0.110,Y -545.353,Z 803.467,A 0.000,B 0.000,C 90.000,E1 120.050} C_DIS
LIN {X -0.126,Y -547.995,Z 803.462,A 0.000,B 0.000,C 90.000,E1 119.205} C_DIS
LIN {X 0.140,Y -551.305,Z 803.456,A 0.000,B 0.000,C 90.000,E1 118.052} C_DIS
LIN {X -0.295,Y -553.518,Z 803.451,A 0.000,B 0.000,C 90.000,E1 117.257} C_DIS
LIN {X 0.273,Y -555.418,Z 803.447,A 0.000,B 0.000,C 90.000,E1 116.360} C_DIS
LIN {X -0.092,Y -557.302,Z 803.440,A 0.000,B 0.000,C 90.000,E1 115.283} C_DIS
LIN {X -0.011,Y -558.211,Z 803.437,A 0.000,B 0.000,C 90.000,E1 114.719} C_DIS
LIN {X 0.174,Y -559.590,Z 803.431,A 0.000,B 0.000,C 90.000,E1 113.590} C_DIS
LIN {X -0.142,Y -560.844,Z 803.425,A 0.000,B 0.000,C 90.000,E1 112.514} C_DIS
LIN {X 0.173,Y -562.208,Z 803.417,A 0.000,B 0.000,C 90.000,E1 111.099} C_DIS
LIN {X -0.211,Y -563.171,Z 803.410,A 0.000,B 0.000,C 90.000,E1 109.758} C_DIS
LIN {X 0.269,Y -563.907,Z 803.401,A 0.000,B 0.000,C 90.000,E1 108.055} C_DIS
LIN {X -0.196,Y -564.818,Z 803.388,A 0.000,B 0.000,C 90.000,E1 105.898} C_DIS
LIN {X -0.004,Y -565.829,Z 803.378,A 0.000,B 0.000,C 90.000,E1 103.953} C_DIS
LIN {X 0.224,Y -567.164,Z 803.367,A 0.000,B 0.000,C 90.000,E1 102.007} C_DIS
LIN {X -0.309,Y -568.531,Z 803.356,A 0.000,B 0.000,C 90.000,E1 100.141} C_DIS
LIN {X -0.055,Y -569.593,Z 803.349,A 0.000,B 0.000,C 90.000,E1 98.746} C_DIS
LIN {X 0.208,Y -570.530,Z 803.341,A 0.000,B 0.000,C 90.000,E1 97.352} C_DIS
LIN {X -0.163,Y -571.367,Z 803.333,A 0.000,B 0.000,C 90.000,E1 96.024} C_DIS
LIN {X 0.247,Y -572.409,Z 803.323,A 0.000,B 0.000,C 90.000,E1 94.073} C_DIS
LIN {X 0.127,Y -573.263,Z 803.312,A 0.000,B 0.000,C 90.000,E1 92.178} C_DIS
LIN {X -0.149,Y -573.856,Z 803.303,A 0.000,B 0.000,C 90.000,E1 90.573} C_DIS
LIN {X 0.147,Y -574.405,Z 803.294,A 0.000,B 0.000,C 90.000,E1 88.912} C_DIS
LIN {X -0.255,Y -574.787,Z 803.287,A 0.000,B 0.000,C 90.000,E1 87.593} C_DIS
LIN {X 0.106,Y -575.162,Z 803.277,A 0.000,B 0.000,C 90.000,E1 85.927} C_DIS
LIN {X -0.291,Y -575.470,Z 803.270,A 0.000,B 0.000,C 90.000,E1 84.609} C_DIS
LIN {X 0.191,Y -575.800,Z 803.261,A 0.000,B 0.000,C 90.000,E1 82.932} C_DIS
LIN {X 0.246,Y -576.183,Z 803.250,A 0.000,B 0.000,C 90.000,E1 81.027} C_DIS
LIN {X 0.270,Y -576.493,Z 803.241,A 0.000,B 0.000,C 90.000,E1 79.398} C_DIS
LIN {X 0.201,Y -576.708,Z 803.234,A 0.000,B 0.000,C 90.000,E1 78.049} C_DIS
LIN {X -0.211,Y -576.717,Z 803.225,A 0.000,B 0.000,C 90.000,E1 76.464} C_DIS
LIN {X 0.065,Y -576.669,Z 803.219,A 0.000,B 0.000,C 90.000,E1 75.353} C_DIS
LIN {X 0.281,Y -576.504,Z 803.211,A 0.000,B 0.000,C 90.000,E1 73.976} C_DIS
LIN {X -0.045,Y -576.322,Z 803.204,A 0.000,B 0.000,C 90.000,E1 72.653} C_DIS
LIN {X 0.174,Y -576.050,Z 803.196,A 0.000,B 0.000,C 90.000,E1 71.275} C_DIS
LIN {X 0.198,Y -575.544,Z 803.187,A 0.000,B 0.000,C 90.000,E1 69.645} C_DIS
LIN {X -0.135,Y -575.113,Z 803.181,A 0.000,B 0.000,C 90.000,E1 68.592} C_DIS
LIN {X -0.095,Y -574.527,Z 803.174,A 0.000,B 0.000,C 90.000,E1 67.230} C_DIS
LIN {X -0.072,Y -573.784,Z 803.166,A 0.000,B 0.000,C 90.000,E1 65.869} C_DIS
LIN {X -0.355,Y -572.995,Z 803.158,A 0.000,B 0.000,C 90.000,E1 64.537} C_DIS
LIN {X 0.117,Y -572.023,Z 803.151,A 0.000,B 0.000,C 90.000,E1 63.127} C_DIS
LIN {X 0.231,Y -571.024,Z 803.145,A 0.000,B 0.000,C 90.000,E1 62.025} C_DIS
LIN {X 0.155,Y -569.491,Z 803.137,A 0.000,B 0.000,C 90.000,E1 60.667} C_DIS
LIN {X 0.016,Y -568.072,Z 803.131,A 0.000,B 0.000,C 90.000,E1 59.587} C_DIS
LIN {X 0.055,Y -566.369,Z 803.125,A 0.000,B 0.000,C 90.000,E1 58.486} C_DIS
LIN {X 0.071,Y -564.965,Z 803.120,A 0.000,B 0.000,C 90.000,E1 57.661} C_DIS
LIN {X 0.078,Y -563.394,Z 803.116,A 0.000,B 0.000,C 90.000,E1 56.834} C_DIS
LIN {X 0.070,Y -561.677,Z 803.111,A 0.000,B 0.000,C 90.000,E1 56.008} C_DIS
LIN {X 0.136,Y -559.015,Z 803.105,A 0.000,B 0.000,C 90.000,E1 54.895} C_DIS
LIN {X 0.076,Y -556.807,Z 803.100,A 0.000,B 0.000,C 90.000,E1 54.069} C_DIS
LIN {X 0.239,Y -555.254,Z 803.097,A 0.000,B 0.000,C 90.000,E1 53.497} C_DIS
LIN {X 0.022,Y -552.604,Z 803.093,A 0.000,B 0.000,C 90.000,E1 52.683} C_DIS
LIN {X 0.218,Y -549.618,Z 803.088,A 0.000,B 0.000,C 90.000,E1 51.823} C_DIS
LIN {X -0.099,Y -547.534,Z 803.085,A 0.000,B 0.000,C 90.000,E1 51.295} C_DIS
LIN {X 0.227,Y -543.334,Z 803.079,A 0.000,B 0.000,C 90.000,E1 50.275} C_DIS
LIN {X -0.130,Y -540.790,Z 803.076,A 0.000,B 0.000,C 90.000,E1 49.747} C_DIS
LIN {X 0.085,Y -537.194,Z 803.072,A 0.000,B 0.000,C 90.000,E1 49.013} C_DIS
LIN {X 0.040,Y -534.090,Z 803.069,A 0.000,B 0.000,C 90.000,E1 48.447} C_DIS
LIN {X 0.015,Y -530.597,Z 803.066,A 0.000,B 0.000,C 90.000,E1 47.877} C_DIS
LIN {X -0.073,Y -526.752,Z 803.063,A 0.000,B 0.000,C 90.000,E1 47.310} C_DIS
LIN {X -0.032,Y -521.335,Z 803.059,A 0.000,B 0.000,C 90.000,E1 46.581} C_DIS
LIN {X 0.054,Y -517.853,Z 803.056,A 0.000,B 0.000,C 90.000,E1 46.134} C_DIS
LIN {X -0.253,Y -514.102,Z 803.054,A 0.000,B 0.000,C 90.000,E1 45.729} C_DIS
LIN {X -0.232,Y -508.852,Z 803.051,A 0.000,B 0.000,C 90.000,E1 45.162} C_DIS
LIN {X -0.255,Y -504.884,Z 803.049,A 0.000,B 0.000,C 90.000,E1 44.757} C_DIS
LIN {X -0.092,Y -499.071,Z 803.045,A 0.000,B 0.000,C 90.000,E1 44.190} C_DIS
LIN {X 0.116,Y -492.021,Z 803.042,A 0.000,B 0.000,C 90.000,E1 43.542} C_DIS
LIN {X -0.052,Y -485.888,Z 803.039,A 0.000,B 0.000,C 90.000,E1 43.056} C_DIS
LIN {X 0.000,Y -479.571,Z 803.037,A 0.000,B 0.000,C 90.000,E1 42.567} C_DIS
LIN {X -0.016,Y -470.020,Z 803.033,A 0.000,B 0.000,C 90.000,E1 41.881} C_DIS
LIN {X -0.019,Y -457.253,Z 803.028,A 0.000,B 0.000,C 90.000,E1 40.987} C_DIS
LIN {X -0.059,Y -442.813,Z 803.022,A 0.000,B 0.000,C 90.000,E1 39.967} C_DIS
LIN {X 0.117,Y -425.600,Z 803.015,A 0.000,B 0.000,C 90.000,E1 38.669} C_DIS
LIN {X 0.059,Y -408.648,Z 803.007,A 0.000,B 0.000,C 90.000,E1 37.282} C_DIS
LIN {X 0.143,Y -404.431,Z 803.005,A 0.000,B 0.000,C 90.000,E1 36.870} C_DIS
LIN {X 0.114,Y -401.830,Z 803.003,A 0.000,B 0.000,C 90.000,E1 36.583} C_DIS
LIN {X 0.085,Y -401.802,Z 803.003,A 0.000,B 0.000,C 90.000,E1 36.583} C_DIS
LIN {X -0.099,Y -394.410,Z 802.979,A 0.000,B 0.000,C 90.000,E1 32.291} C_DIS
LIN {X 0.107,Y -394.255,Z 802.978,A 0.000,B 0.000,C 90.000,E1 32.084} C_DIS
LIN {X -0.088,Y -395.258,Z 802.964,A 0.000,B 0.000,C 90.000,E1 29.461} C_DIS
LIN {X -0.164,Y -396.572,Z 802.950,A 0.000,B 0.000,C 90.000,E1 27.001} C_DIS
LIN {X 0.058,Y -397.642,Z 802.940,A 0.000,B 0.000,C 90.000,E1 25.207} C_DIS
LIN {X -0.033,Y -398.814,Z 802.930,A 0.000,B 0.000,C 90.000,E1 23.462} C_DIS
LIN {X 0.088,Y -401.704,Z 802.911,A 0.000,B 0.000,C 90.000,E1 19.939} C_DIS
LIN {X 0.062,Y -405.100,Z 802.893,A 0.000,B 0.000,C 90.000,E1 16.804} C_DIS
LIN {X -0.076,Y -409.491,Z 802.876,A 0.000,B 0.000,C 90.000,E1 13.703} C_DIS
LIN {X -0.124,Y -413.416,Z 802.863,A 0.000,B 0.000,C 90.000,E1 11.299} C_DIS
LIN {X 0.198,Y -417.586,Z 802.849,A 0.000,B 0.000,C 90.000,E1 8.859} C_DIS
LIN {X 0.028,Y -420.680,Z 802.840,A 0.000,B 0.000,C 90.000,E1 7.182} C_DIS
LIN {X -0.016,Y -424.999,Z 802.827,A 0.000,B 0.000,C 90.000,E1 4.821} C_DIS
LIN {X 0.092,Y -430.102,Z 802.812,A 0.000,B 0.000,C 90.000,E1 2.121} C_DIS
LIN {X -0.178,Y -435.594,Z 802.797,A 0.000,B 0.000,C 90.000,E1 359.484} C_DIS
LIN {X 0.117,Y -440.745,Z 802.784,A 0.000,B 0.000,C 90.000,E1 357.135} C_DIS
LIN {X 0.164,Y -446.252,Z 802.771,A 0.000,B 0.000,C 90.000,E1 354.837} C_DIS
LIN {X -0.184,Y -451.042,Z 802.761,A 0.000,B 0.000,C 90.000,E1 352.932} C_DIS
LIN {X -0.123,Y -454.957,Z 802.752,A 0.000,B 0.000,C 90.000,E1 351.310} C_DIS
LIN {X -0.219,Y -458.237,Z 802.745,A 0.000,B 0.000,C 90.000,E1 350.038} C_DIS
LIN {X 0.039,Y -461.355,Z 802.739,A 0.000,B 0.000,C 90.000,E1 349.050} C_DIS
LIN {X -0.006,Y -463.609,Z 802.737,A 0.000,B 0.000,C 90.000,E1 348.578} C_DIS
LIN {X -0.162,Y -465.920,Z 802.735,A 0.000,B 0.000,C 90.000,E1 348.229} C_DIS
LIN {X -0.126,Y -469.982,Z 802.732,A 0.000,B 0.000,C 90.000,E1 347.757} C_DIS
LIN {X 0.017,Y -474.031,Z 802.730,A 0.000,B 0.000,C 90.000,E1 347.353} C_DIS
LIN {X 0.002,Y -479.681,Z 802.727,A 0.000,B 0.000,C 90.000,E1 346.881} C_DIS
LIN {X -0.146,Y -495.016,Z 802.721,A 0.000,B 0.000,C 90.000,E1 345.811} C_DIS
LIN {X 0.152,Y -513.696,Z 802.714,A 0.000,B 0.000,C 90.000,E1 344.519} C_DIS
LIN {X -0.126,Y -527.515,Z 802.709,A 0.000,B 0.000,C 90.000,E1 343.614} C_DIS
LIN {X -0.072,Y -536.672,Z 802.705,A 0.000,B 0.000,C 90.000,E1 342.960} C_DIS
LIN {X -0.292,Y -542.650,Z 802.703,A 0.000,B 0.000,C 90.000,E1 342.543} C_DIS
LIN {X -0.265,Y -549.898,Z 802.700,A 0.000,B 0.000,C 90.000,E1 342.000} C_DIS
LIN {X 0.107,Y -553.997,Z 802.698,A 0.000,B 0.000,C 90.000,E1 341.638} C_DIS
LIN {X 0.197,Y -559.481,Z 802.695,A 0.000,B 0.000,C 90.000,E1 341.148} C_DIS
LIN {X -0.034,Y -564.951,Z 802.693,A 0.000,B 0.000,C 90.000,E1 340.678} C_DIS
LIN {X -0.259,Y -570.134,Z 802.690,A 0.000,B 0.000,C 90.000,E1 340.188} C_DIS
LIN {X 0.021,Y -574.983,Z 802.687,A 0.000,B 0.000,C 90.000,E1 339.625} C_DIS
LIN {X -0.057,Y -580.506,Z 802.683,A 0.000,B 0.000,C 90.000,E1 338.954} C_DIS
LIN {X -0.022,Y -584.591,Z 802.680,A 0.000,B 0.000,C 90.000,E1 338.411} C_DIS
LIN {X -0.087,Y -590.355,Z 802.676,A 0.000,B 0.000,C 90.000,E1 337.614} C_DIS
LIN {X 0.187,Y -594.820,Z 802.672,A 0.000,B 0.000,C 90.000,E1 336.922} C_DIS
LIN {X 0.071,Y -603.295,Z 802.665,A 0.000,B 0.000,C 90.000,E1 335.613} C_DIS
LIN {X -0.160,Y -609.656,Z 802.659,A 0.000,B 0.000,C 90.000,E1 334.588} C_DIS
LIN {X 0.278,Y -614.204,Z 802.654,A 0.000,B 0.000,C 90.000,E1 333.768} C_DIS
LIN {X 0.193,Y -620.651,Z 802.648,A 0.000,B 0.000,C 90.000,E1 332.615} C_DIS
LIN {X 0.187,Y -624.791,Z 802.644,A 0.000,B 0.000,C 90.000,E1 331.847} C_DIS
LIN {X -0.021,Y -629.172,Z 802.639,A 0.000,B 0.000,C 90.000,E1 330.973} C_DIS
LIN {X 0.098,Y -634.844,Z 802.632,A 0.000,B 0.000,C 90.000,E1 329.822} C_DIS
LIN {X 0.029,Y -639.509,Z 802.627,A 0.000,B 0.000,C 90.000,E1 328.820} C_DIS
LIN {X -0.037,Y -642.778,Z 802.623,A 0.000,B 0.000,C 90.000,E1 328.074} C_DIS
LIN {X -0.070,Y -648.877,Z 802.614,A 0.000,B 0.000,C 90.000,E1 326.580} C_DIS
LIN {X 0.321,Y -651.685,Z 802.610,A 0.000,B 0.000,C 90.000,E1 325.801} C_DIS
LIN {X -0.084,Y -655.194,Z 802.605,A 0.000,B 0.000,C 90.000,E1 324.848} C_DIS
LIN {X -0.075,Y -658.377,Z 802.599,A 0.000,B 0.000,C 90.000,E1 323.863} C_DIS
LIN {X 0.371,Y -661.428,Z 802.594,A 0.000,B 0.000,C 90.000,E1 322.844} C_DIS
LIN {X -0.066,Y -664.286,Z 802.588,A 0.000,B 0.000,C 90.000,E1 321.904} C_DIS
LIN {X 0.029,Y -667.562,Z 802.582,A 0.000,B 0.000,C 90.000,E1 320.678} C_DIS
LIN {X 0.082,Y -670.499,Z 802.575,A 0.000,B 0.000,C 90.000,E1 319.461} C_DIS
LIN {X 0.190,Y -673.227,Z 802.568,A 0.000,B 0.000,C 90.000,E1 318.243} C_DIS
LIN {X -0.206,Y -674.784,Z 802.564,A 0.000,B 0.000,C 90.000,E1 317.553} C_DIS
LIN {X -0.066,Y -677.049,Z 802.557,A 0.000,B 0.000,C 90.000,E1 316.338} C_DIS
LIN {X 0.054,Y -678.343,Z 802.553,A 0.000,B 0.000,C 90.000,E1 315.607} C_DIS
LIN {X -0.184,Y -680.476,Z 802.545,A 0.000,B 0.000,C 90.000,E1 314.190} C_DIS
LIN {X 0.045,Y -682.149,Z 802.539,A 0.000,B 0.000,C 90.000,E1 312.975} C_DIS
LIN {X 0.284,Y -683.399,Z 802.534,A 0.000,B 0.000,C 90.000,E1 312.000} C_DIS
LIN {X 0.087,Y -684.866,Z 802.527,A 0.000,B 0.000,C 90.000,E1 310.825} C_DIS
LIN {X -0.072,Y -685.925,Z 802.522,A 0.000,B 0.000,C 90.000,E1 309.886} C_DIS
LIN {X -0.102,Y -687.376,Z 802.514,A 0.000,B 0.000,C 90.000,E1 308.463} C_DIS
LIN {X 0.049,Y -688.892,Z 802.504,A 0.000,B 0.000,C 90.000,E1 306.790} C_DIS
LIN {X 0.142,Y -689.899,Z 802.498,A 0.000,B 0.000,C 90.000,E1 305.598} C_DIS
LIN {X -0.106,Y -691.002,Z 802.490,A 0.000,B 0.000,C 90.000,E1 304.199} C_DIS
LIN {X -0.122,Y -692.207,Z 802.481,A 0.000,B 0.000,C 90.000,E1 302.546} C_DIS
LIN {X 0.105,Y -693.456,Z 802.472,A 0.000,B 0.000,C 90.000,E1 300.875} C_DIS
LIN {X -0.132,Y -694.281,Z 802.465,A 0.000,B 0.000,C 90.000,E1 299.716} C_DIS
LIN {X 0.139,Y -695.143,Z 802.457,A 0.000,B 0.000,C 90.000,E1 298.281} C_DIS
LIN {X -0.002,Y -696.335,Z 802.447,A 0.000,B 0.000,C 90.000,E1 296.411} C_DIS
LIN {X -0.052,Y -697.540,Z 802.438,A 0.000,B 0.000,C 90.000,E1 294.771} C_DIS
LIN {X 0.181,Y -697.704,Z 802.435,A 0.000,B 0.000,C 90.000,E1 294.283} C_DIS
LIN {X 0.065,Y -697.340,Z 802.432,A 0.000,B 0.000,C 90.000,E1 293.823} C_DIS
LIN {X 0.044,Y -697.075,Z 802.431,A 0.000,B 0.000,C 90.000,E1 293.590} C_DIS
LIN {X 0.302,Y -696.264,Z 802.430,A 0.000,B 0.000,C 90.000,E1 293.334} C_DIS
LIN {X -0.229,Y -694.590,Z 802.428,A 0.000,B 0.000,C 90.000,E1 293.025} C_DIS
LIN {X -0.103,Y -693.955,Z 802.427,A 0.000,B 0.000,C 90.000,E1 292.898} C_DIS
LIN {X 0.020,Y -693.056,Z 802.427,A 0.000,B 0.000,C 90.000,E1 292.770} C_DIS
LIN {X 0.142,Y -691.720,Z 802.426,A 0.000,B 0.000,C 90.000,E1 292.642} C_DIS
LIN {X -0.362,Y -688.426,Z 802.425,A 0.000,B 0.000,C 90.000,E1 292.461} C_DIS
LIN {X 0.385,Y -685.101,Z 802.424,A 0.000,B 0.000,C 90.000,E1 292.206} C_DIS
LIN {X -0.012,Y -683.107,Z 802.423,A 0.000,B 0.000,C 90.000,E1 292.153} C_DIS
LIN {X -0.203,Y -678.595,Z 802.422,A 0.000,B 0.000,C 90.000,E1 292.025} C_DIS
LIN {X 0.063,Y -673.172,Z 802.421,A 0.000,B 0.000,C 90.000,E1 291.844} C_DIS
LIN {X -0.358,Y -663.958,Z 802.421,A 0.000,B 0.000,C 90.000,E1 291.716} C_DIS
LIN {X -0.103,Y -645.996,Z 802.419,A 0.000,B 0.000,C 90.000,E1 291.408} C_DIS
LIN {X -0.088,Y -631.974,Z 802.418,A 0.000,B 0.000,C 90.000,E1 291.153} C_DIS
LIN {X -0.081,Y -618.393,Z 802.416,A 0.000,B 0.000,C 90.000,E1 290.865} C_DIS
LIN {X -0.022,Y -608.391,Z 802.415,A 0.000,B 0.000,C 90.000,E1 290.610} C_DIS
LIN {X -0.042,Y -602.007,Z 802.414,A 0.000,B 0.000,C 90.000,E1 290.429} C_DIS
LIN {X 0.103,Y -589.482,Z 802.411,A 0.000,B 0.000,C 90.000,E1 289.993} C_DIS
LIN {X -0.064,Y -586.009,Z 802.410,A 0.000,B 0.000,C 90.000,E1 289.885} C_DIS
LIN {X 0.034,Y -580.424,Z 802.409,A 0.000,B 0.000,C 90.000,E1 289.631} C_DIS
LIN {X 0.182,Y -578.126,Z 802.409,A 0.000,B 0.000,C 90.000,E1 289.504} C_DIS
LIN {X -0.202,Y -576.418,Z 802.408,A 0.000,B 0.000,C 90.000,E1 289.396} C_DIS
LIN {X -0.068,Y -574.509,Z 802.407,A 0.000,B 0.000,C 90.000,E1 289.268} C_DIS
LIN {X 0.063,Y -572.887,Z 802.406,A 0.000,B 0.000,C 90.000,E1 289.141} C_DIS
LIN {X 0.252,Y -572.248,Z 802.406,A 0.000,B 0.000,C 90.000,E1 288.960} C_DIS
LIN {X 0.210,Y -572.088,Z 802.403,A 0.000,B 0.000,C 90.000,E1 288.544} C_DIS
LIN {X 0.117,Y -572.413,Z 802.402,A 0.000,B 0.000,C 90.000,E1 288.417} C_DIS
LIN {X 0.102,Y -575.211,Z 802.399,A 0.000,B 0.000,C 90.000,E1 287.873} C_DIS
LIN {X -0.247,Y -580.203,Z 802.395,A 0.000,B 0.000,C 90.000,E1 287.094} C_DIS
LIN {X -0.076,Y -585.043,Z 802.390,A 0.000,B 0.000,C 90.000,E1 286.134} C_DIS
LIN {X -0.170,Y -587.621,Z 802.387,A 0.000,B 0.000,C 90.000,E1 285.607} C_DIS
LIN {X 0.165,Y -590.585,Z 802.382,A 0.000,B 0.000,C 90.000,E1 284.773} C_DIS
LIN {X -0.149,Y -591.144,Z 802.381,A 0.000,B 0.000,C 90.000,E1 284.537} C_DIS
LIN {X 0.114,Y -591.554,Z 802.379,A 0.000,B 0.000,C 90.000,E1 284.245} C_DIS
LIN {X 0.075,Y -592.002,Z 802.376,A 0.000,B 0.000,C 90.000,E1 283.716} C_DIS
LIN {X -0.092,Y -592.139,Z 802.375,A 0.000,B 0.000,C 90.000,E1 283.467} C_DIS
LIN {X -0.129,Y -591.785,Z 802.372,A 0.000,B 0.000,C 90.000,E1 282.939} C_DIS
LIN {X -0.167,Y -590.935,Z 802.369,A 0.000,B 0.000,C 90.000,E1 282.411} C_DIS
LIN {X -0.210,Y -589.584,Z 802.366,A 0.000,B 0.000,C 90.000,E1 281.883} C_DIS
LIN {X 0.055,Y -588.736,Z 802.365,A 0.000,B 0.000,C 90.000,E1 281.591} C_DIS
LIN {X -0.116,Y -586.433,Z 802.362,A 0.000,B 0.000,C 90.000,E1 281.074} C_DIS
LIN {X -0.188,Y -583.375,Z 802.359,A 0.000,B 0.000,C 90.000,E1 280.546} C_DIS
LIN {X 0.052,Y -581.316,Z 802.357,A 0.000,B 0.000,C 90.000,E1 280.254} C_DIS
LIN {X 0.285,Y -578.417,Z 802.356,A 0.000,B 0.000,C 90.000,E1 279.962} C_DIS
LIN {X 0.205,Y -576.624,Z 802.355,A 0.000,B 0.000,C 90.000,E1 279.849} C_DIS
LIN {X -0.096,Y -572.683,Z 802.354,A 0.000,B 0.000,C 90.000,E1 279.670} C_DIS
LIN {X 0.218,Y -566.250,Z 802.353,A 0.000,B 0.000,C 90.000,E1 279.443} C_DIS
LIN {X 0.272,Y -560.423,Z 802.351,A 0.000,B 0.000,C 90.000,E1 279.208} C_DIS
LIN {X 0.099,Y -555.246,Z 802.350,A 0.000,B 0.000,C 90.000,E1 278.973} C_DIS
LIN {X 0.278,Y -554.674,Z 802.350,A 0.000,B 0.000,C 90.000,E1 278.916} C_DIS
LIN {X -0.085,Y -551.366,Z 802.347,A 0.000,B 0.000,C 90.000,E1 278.511} C_DIS
LIN {X -0.127,Y -551.332,Z 802.347,A 0.000,B 0.000,C 90.000,E1 278.511} C_DIS
LIN {X 0.059,Y -550.962,Z 802.344,A 0.000,B 0.000,C 90.000,E1 277.814} C_DIS
LIN {X 0.094,Y -550.934,Z 802.342,A 0.000,B 0.000,C 90.000,E1 277.530} C_DIS
LIN {X 0.229,Y -549.740,Z 802.328,A 0.000,B 0.000,C 90.000,E1 274.992} C_DIS
LIN {X -0.001,Y -548.924,Z 802.320,A 0.000,B 0.000,C 90.000,E1 273.612} C_DIS
LIN {X -0.280,Y -547.979,Z 802.312,A 0.000,B 0.000,C 90.000,E1 272.236} C_DIS
LIN {X 0.062,Y -546.637,Z 802.301,A 0.000,B 0.000,C 90.000,E1 270.229} C_DIS
LIN {X 0.235,Y -545.900,Z 802.295,A 0.000,B 0.000,C 90.000,E1 269.083} C_DIS
LIN {X 0.033,Y -544.330,Z 802.283,A 0.000,B 0.000,C 90.000,E1 266.846} C_DIS
LIN {X 0.214,Y -543.437,Z 802.275,A 0.000,B 0.000,C 90.000,E1 265.412} C_DIS
LIN {X -0.131,Y -542.566,Z 802.267,A 0.000,B 0.000,C 90.000,E1 264.033} C_DIS
LIN {X 0.102,Y -541.487,Z 802.259,A 0.000,B 0.000,C 90.000,E1 262.591} C_DIS
LIN {X -0.144,Y -540.251,Z 802.251,A 0.000,B 0.000,C 90.000,E1 261.197} C_DIS
LIN {X 0.056,Y -539.268,Z 802.245,A 0.000,B 0.000,C 90.000,E1 260.038} C_DIS
LIN {X 0.007,Y -537.316,Z 802.234,A 0.000,B 0.000,C 90.000,E1 258.049} C_DIS
LIN {X -0.153,Y -535.604,Z 802.224,A 0.000,B 0.000,C 90.000,E1 256.353} C_DIS
LIN {X -0.099,Y -533.698,Z 802.215,A 0.000,B 0.000,C 90.000,E1 254.629} C_DIS
LIN {X 0.101,Y -531.354,Z 802.203,A 0.000,B 0.000,C 90.000,E1 252.598} C_DIS
LIN {X 0.197,Y -529.623,Z 802.195,A 0.000,B 0.000,C 90.000,E1 251.148} C_DIS
LIN {X 0.256,Y -527.731,Z 802.187,A 0.000,B 0.000,C 90.000,E1 249.699} C_DIS
LIN {X -0.209,Y -526.110,Z 802.181,A 0.000,B 0.000,C 90.000,E1 248.592} C_DIS
LIN {X -0.160,Y -523.554,Z 802.171,A 0.000,B 0.000,C 90.000,E1 246.847} C_DIS
LIN {X 0.155,Y -521.377,Z 802.163,A 0.000,B 0.000,C 90.000,E1 245.357} C_DIS
LIN {X 0.024,Y -519.543,Z 802.157,A 0.000,B 0.000,C 90.000,E1 244.204} C_DIS
LIN {X 0.125,Y -516.519,Z 802.147,A 0.000,B 0.000,C 90.000,E1 242.436} C_DIS
LIN {X 0.161,Y -514.459,Z 802.140,A 0.000,B 0.000,C 90.000,E1 241.257} C_DIS
LIN {X 0.071,Y -511.678,Z 802.132,A 0.000,B 0.000,C 90.000,E1 239.793} C_DIS
LIN {X 0.036,Y -509.372,Z 802.126,A 0.000,B 0.000,C 90.000,E1 238.614} C_DIS
LIN {X -0.103,Y -507.560,Z 802.121,A 0.000,B 0.000,C 90.000,E1 237.740} C_DIS
LIN {X -0.092,Y -505.053,Z 802.114,A 0.000,B 0.000,C 90.000,E1 236.548} C_DIS
LIN {X -0.092,Y -501.830,Z 802.106,A 0.000,B 0.000,C 90.000,E1 235.055} C_DIS
LIN {X -0.039,Y -499.784,Z 802.101,A 0.000,B 0.000,C 90.000,E1 234.149} C_DIS
LIN {X 0.021,Y -496.026,Z 802.092,A 0.000,B 0.000,C 90.000,E1 232.637} C_DIS
LIN {X 0.010,Y -492.211,Z 802.084,A 0.000,B 0.000,C 90.000,E1 231.126} C_DIS
LIN {X -0.042,Y -485.092,Z 802.067,A 0.000,B 0.000,C 90.000,E1 228.081} C_DIS
LIN {X 0.258,Y -480.454,Z 802.055,A 0.000,B 0.000,C 90.000,E1 225.891} C_DIS
LIN {X -0.259,Y -475.652,Z 802.043,A 0.000,B 0.000,C 90.000,E1 223.785} C_DIS
LIN {X -0.171,Y -472.900,Z 802.036,A 0.000,B 0.000,C 90.000,E1 222.528} C_DIS
LIN {X -0.006,Y -469.565,Z 802.028,A 0.000,B 0.000,C 90.000,E1 220.943} C_DIS
LIN {X -0.084,Y -465.001,Z 802.015,A 0.000,B 0.000,C 90.000,E1 218.749} C_DIS
LIN {X -0.257,Y -460.997,Z 802.005,A 0.000,B 0.000,C 90.000,E1 216.870} C_DIS
LIN {X -0.007,Y -459.021,Z 801.999,A 0.000,B 0.000,C 90.000,E1 215.884} C_DIS
LIN {X -0.213,Y -455.078,Z 801.989,A 0.000,B 0.000,C 90.000,E1 213.992} C_DIS
LIN {X -0.055,Y -450.494,Z 801.976,A 0.000,B 0.000,C 90.000,E1 211.720} C_DIS
LIN {X -0.192,Y -446.625,Z 801.965,A 0.000,B 0.000,C 90.000,E1 209.795} C_DIS
LIN {X -0.241,Y -442.772,Z 801.955,A 0.000,B 0.000,C 90.000,E1 207.847} C_DIS
LIN {X -0.021,Y -439.708,Z 801.945,A 0.000,B 0.000,C 90.000,E1 206.181} C_DIS
LIN {X -0.035,Y -435.926,Z 801.935,A 0.000,B 0.000,C 90.000,E1 204.207} C_DIS
LIN {X -0.143,Y -433.297,Z 801.927,A 0.000,B 0.000,C 90.000,E1 202.898} C_DIS
LIN {X 0.138,Y -429.462,Z 801.916,A 0.000,B 0.000,C 90.000,E1 200.865} C_DIS
LIN {X -0.031,Y -424.995,Z 801.903,A 0.000,B 0.000,C 90.000,E1 198.544} C_DIS
LIN {X -0.022,Y -421.730,Z 801.894,A 0.000,B 0.000,C 90.000,E1 196.858} C_DIS
LIN {X 0.151,Y -419.136,Z 801.886,A 0.000,B 0.000,C 90.000,E1 195.481} C_DIS
LIN {X -0.044,Y -415.189,Z 801.875,A 0.000,B 0.000,C 90.000,E1 193.467} C_DIS
LIN {X -0.150,Y -412.005,Z 801.865,A 0.000,B 0.000,C 90.000,E1 191.771} C_DIS
LIN {X 0.133,Y -407.720,Z 801.852,A 0.000,B 0.000,C 90.000,E1 189.321} C_DIS
LIN {X 0.138,Y -405.222,Z 801.844,A 0.000,B 0.000,C 90.000,E1 187.936} C_DIS
LIN {X 0.100,Y -401.386,Z 801.833,A 0.000,B 0.000,C 90.000,E1 185.853} C_DIS
LIN {X -0.120,Y -394.245,Z 801.807,A 0.000,B 0.000,C 90.000,E1 181.318} C_DIS
LIN {X 0.157,Y -391.268,Z 801.794,A 0.000,B 0.000,C 90.000,E1 178.797} C_DIS
LIN {X 0.140,Y -389.357,Z 801.784,A 0.000,B 0.000,C 90.000,E1 177.020} C_DIS
LIN {X -0.037,Y -386.670,Z 801.770,A 0.000,B 0.000,C 90.000,E1 174.546} C_DIS
LIN {X -0.090,Y -384.793,Z 801.760,A 0.000,B 0.000,C 90.000,E1 172.761} C_DIS
LIN {X -0.144,Y -383.075,Z 801.750,A 0.000,B 0.000,C 90.000,E1 170.971} C_DIS
LIN {X 0.089,Y -380.861,Z 801.736,A 0.000,B 0.000,C 90.000,E1 168.409} C_DIS
LIN {X 0.031,Y -378.654,Z 801.720,A 0.000,B 0.000,C 90.000,E1 165.519} C_DIS
LIN {X 0.132,Y -377.330,Z 801.708,A 0.000,B 0.000,C 90.000,E1 163.323} C_DIS
LIN {X -0.020,Y -376.048,Z 801.685,A 0.000,B 0.000,C 90.000,E1 159.337} C_DIS
LIN {X -0.121,Y -376.408,Z 801.661,A 0.000,B 0.000,C 90.000,E1 154.973} C_DIS
LIN {X 0.025,Y -377.312,Z 801.651,A 0.000,B 0.000,C 90.000,E1 153.127} C_DIS
LIN {X -0.025,Y -379.779,Z 801.637,A 0.000,B 0.000,C 90.000,E1 150.589} C_DIS
LIN {X 0.065,Y -381.513,Z 801.631,A 0.000,B 0.000,C 90.000,E1 149.488} C_DIS
LIN {X 0.039,Y -383.734,Z 801.625,A 0.000,B 0.000,C 90.000,E1 148.408} C_DIS
LIN {X -0.110,Y -385.544,Z 801.621,A 0.000,B 0.000,C 90.000,E1 147.709} C_DIS
LIN {X -0.082,Y -388.901,Z 801.615,A 0.000,B 0.000,C 90.000,E1 146.628} C_DIS
LIN {X -0.051,Y -390.739,Z 801.612,A 0.000,B 0.000,C 90.000,E1 146.087} C_DIS
LIN {X -0.136,Y -393.640,Z 801.608,A 0.000,B 0.000,C 90.000,E1 145.388} C_DIS
LIN {X -0.082,Y -396.166,Z 801.605,A 0.000,B 0.000,C 90.000,E1 144.848} C_DIS
LIN {X -0.148,Y -401.132,Z 801.600,A 0.000,B 0.000,C 90.000,E1 143.989} C_DIS
LIN {X -0.051,Y -404.405,Z 801.597,A 0.000,B 0.000,C 90.000,E1 143.463} C_DIS
LIN {X -0.101,Y -411.821,Z 801.591,A 0.000,B 0.000,C 90.000,E1 142.477} C_DIS
LIN {X -0.075,Y -418.326,Z 801.587,A 0.000,B 0.000,C 90.000,E1 141.662} C_DIS
LIN {X -0.150,Y -423.802,Z 801.583,A 0.000,B 0.000,C 90.000,E1 141.009} C_DIS
LIN {X -0.091,Y -427.671,Z 801.581,A 0.000,B 0.000,C 90.000,E1 140.517} C_DIS
LIN {X -0.004,Y -436.708,Z 801.574,A 0.000,B 0.000,C 90.000,E1 139.337} C_DIS
LIN {X -0.136,Y -453.416,Z 801.562,A 0.000,B 0.000,C 90.000,E1 137.229} C_DIS
LIN {X -0.115,Y -457.169,Z 801.560,A 0.000,B 0.000,C 90.000,E1 136.743} C_DIS
LIN {X 0.006,Y -464.031,Z 801.554,A 0.000,B 0.000,C 90.000,E1 135.769} C_DIS
LIN {X 0.031,Y -474.547,Z 801.546,A 0.000,B 0.000,C 90.000,E1 134.190} C_DIS
LIN {X -0.040,Y -479.851,Z 801.541,A 0.000,B 0.000,C 90.000,E1 133.419} C_DIS
LIN {X 0.012,Y -485.912,Z 801.536,A 0.000,B 0.000,C 90.000,E1 132.486} C_DIS
LIN {X 0.304,Y -489.683,Z 801.533,A 0.000,B 0.000,C 90.000,E1 131.838} C_DIS
LIN {X 0.151,Y -497.550,Z 801.525,A 0.000,B 0.000,C 90.000,E1 130.539} C_DIS
LIN {X 0.173,Y -503.601,Z 801.520,A 0.000,B 0.000,C 90.000,E1 129.483} C_DIS
LIN {X -0.011,Y -509.333,Z 801.514,A 0.000,B 0.000,C 90.000,E1 128.463} C_DIS
LIN {X -0.160,Y -514.715,Z 801.508,A 0.000,B 0.000,C 90.000,E1 127.443} C_DIS
LIN {X 0.234,Y -518.377,Z 801.504,A 0.000,B 0.000,C 90.000,E1 126.664} C_DIS
LIN {X 0.021,Y -524.022,Z 801.497,A 0.000,B 0.000,C 90.000,E1 125.518} C_DIS
LIN {X -0.228,Y -527.213,Z 801.493,A 0.000,B 0.000,C 90.000,E1 124.818} C_DIS
LIN {X -0.212,Y -533.109,Z 801.485,A 0.000,B 0.000,C 90.000,E1 123.372} C_DIS
LIN {X -0.091,Y -537.588,Z 801.479,A 0.000,B 0.000,C 90.000,E1 122.212} C_DIS
LIN {X 0.090,Y -541.807,Z 801.473,A 0.000,B 0.000,C 90.000,E1 121.052} C_DIS
LIN {X 0.033,Y -544.701,Z 801.468,A 0.000,B 0.000,C 90.000,E1 120.207} C_DIS
LIN {X 0.285,Y -547.406,Z 801.463,A 0.000,B 0.000,C 90.000,E1 119.333} C_DIS
LIN {X -0.180,Y -551.535,Z 801.455,A 0.000,B 0.000,C 90.000,E1 117.975} C_DIS
LIN {X -0.124,Y -553.744,Z 801.451,A 0.000,B 0.000,C 90.000,E1 117.129} C_DIS
LIN {X -0.050,Y -555.604,Z 801.446,A 0.000,B 0.000,C 90.000,E1 116.283} C_DIS
LIN {X -0.127,Y -558.018,Z 801.438,A 0.000,B 0.000,C 90.000,E1 114.899} C_DIS
LIN {X -0.252,Y -559.143,Z 801.434,A 0.000,B 0.000,C 90.000,E1 114.079} C_DIS
LIN {X 0.248,Y -560.700,Z 801.426,A 0.000,B 0.000,C 90.000,E1 112.642} C_DIS
LIN {X 0.040,Y -562.087,Z 801.418,A 0.000,B 0.000,C 90.000,E1 111.280} C_DIS
LIN {X 0.181,Y -563.132,Z 801.411,A 0.000,B 0.000,C 90.000,E1 109.885} C_DIS
LIN {X 0.210,Y -563.672,Z 801.404,A 0.000,B 0.000,C 90.000,E1 108.779} C_DIS
LIN {X 0.056,Y -564.170,Z 801.398,A 0.000,B 0.000,C 90.000,E1 107.692} C_DIS
LIN {X -0.173,Y -565.056,Z 801.388,A 0.000,B 0.000,C 90.000,E1 105.788} C_DIS
LIN {X -0.039,Y -566.521,Z 801.374,A 0.000,B 0.000,C 90.000,E1 103.300} C_DIS
LIN {X -0.097,Y -567.659,Z 801.365,A 0.000,B 0.000,C 90.000,E1 101.658} C_DIS
LIN {X 0.041,Y -569.087,Z 801.354,A 0.000,B 0.000,C 90.000,E1 99.726} C_DIS
LIN {X 0.112,Y -569.939,Z 801.348,A 0.000,B 0.000,C 90.000,E1 98.624} C_DIS
LIN {X -0.266,Y -570.876,Z 801.340,A 0.000,B 0.000,C 90.000,E1 97.296} C_DIS
LIN {X 0.059,Y -571.896,Z 801.331,A 0.000,B 0.000,C 90.000,E1 95.625} C_DIS
LIN {X -0.170,Y -572.751,Z 801.322,A 0.000,B 0.000,C 90.000,E1 94.012} C_DIS
LIN {X 0.251,Y -573.609,Z 801.312,A 0.000,B 0.000,C 90.000,E1 92.064} C_DIS
LIN {X -0.163,Y -574.114,Z 801.304,A 0.000,B 0.000,C 90.000,E1 90.745} C_DIS
LIN {X -0.289,Y -574.743,Z 801.294,A 0.000,B 0.000,C 90.000,E1 88.854} C_DIS
LIN {X -0.111,Y -575.130,Z 801.286,A 0.000,B 0.000,C 90.000,E1 87.478} C_DIS
LIN {X 0.257,Y -575.520,Z 801.277,A 0.000,B 0.000,C 90.000,E1 85.812} C_DIS
LIN {X 0.056,Y -575.891,Z 801.268,A 0.000,B 0.000,C 90.000,E1 84.204} C_DIS
LIN {X 0.112,Y -576.260,Z 801.257,A 0.000,B 0.000,C 90.000,E1 82.299} C_DIS
LIN {X 0.257,Y -576.635,Z 801.247,A 0.000,B 0.000,C 90.000,E1 80.387} C_DIS
LIN {X 0.079,Y -576.902,Z 801.239,A 0.000,B 0.000,C 90.000,E1 79.050} C_DIS
LIN {X 0.014,Y -577.017,Z 801.232,A 0.000,B 0.000,C 90.000,E1 77.701} C_DIS
LIN {X 0.162,Y -576.966,Z 801.223,A 0.000,B 0.000,C 90.000,E1 76.061} C_DIS
LIN {X 0.022,Y -576.874,Z 801.217,A 0.000,B 0.000,C 90.000,E1 74.991} C_DIS
LIN {X -0.103,Y -576.645,Z 801.208,A 0.000,B 0.000,C 90.000,E1 73.378} C_DIS
LIN {X 0.123,Y -576.396,Z 801.200,A 0.000,B 0.000,C 90.000,E1 72.000} C_DIS
LIN {X -0.223,Y -576.223,Z 801.196,A 0.000,B 0.000,C 90.000,E1 71.221} C_DIS
LIN {X 0.000,Y -575.696,Z 801.187,A 0.000,B 0.000,C 90.000,E1 69.571} C_DIS
LIN {X -0.163,Y -575.122,Z 801.179,A 0.000,B 0.000,C 90.000,E1 68.230} C_DIS
LIN {X -0.129,Y -574.488,Z 801.171,A 0.000,B 0.000,C 90.000,E1 66.869} C_DIS
LIN {X 0.120,Y -573.672,Z 801.164,A 0.000,B 0.000,C 90.000,E1 65.485} C_DIS
LIN {X -0.001,Y -573.014,Z 801.158,A 0.000,B 0.000,C 90.000,E1 64.409} C_DIS
LIN {X -0.039,Y -571.981,Z 801.150,A 0.000,B 0.000,C 90.000,E1 63.050} C_DIS
LIN {X -0.190,Y -570.963,Z 801.144,A 0.000,B 0.000,C 90.000,E1 61.975} C_DIS
LIN {X 0.180,Y -569.700,Z 801.138,A 0.000,B 0.000,C 90.000,E1 60.845} C_DIS
LIN {X -0.059,Y -568.652,Z 801.134,A 0.000,B 0.000,C 90.000,E1 60.049} C_DIS
LIN {X -0.007,Y -567.024,Z 801.128,A 0.000,B 0.000,C 90.000,E1 58.948} C_DIS
LIN {X -0.178,Y -565.221,Z 801.121,A 0.000,B 0.000,C 90.000,E1 57.867} C_DIS
LIN {X -0.065,Y -563.047,Z 801.115,A 0.000,B 0.000,C 90.000,E1 56.755} C_DIS
LIN {X -0.074,Y -561.297,Z 801.111,A 0.000,B 0.000,C 90.000,E1 55.928} C_DIS
LIN {X -0.103,Y -559.259,Z 801.106,A 0.000,B 0.000,C 90.000,E1 55.102} C_DIS
LIN {X -0.158,Y -557.077,Z 801.102,A 0.000,B 0.000,C 90.000,E1 54.276} C_DIS
LIN {X 0.086,Y -554.623,Z 801.097,A 0.000,B 0.000,C 90.000,E1 53.417} C_DIS
LIN {X 0.304,Y -551.869,Z 801.092,A 0.000,B 0.000,C 90.000,E1 52.557} C_DIS
LIN {X -0.002,Y -549.913,Z 801.089,A 0.000,B 0.000,C 90.000,E1 52.029} C_DIS
LIN {X 0.161,Y -546.663,Z 801.084,A 0.000,B 0.000,C 90.000,E1 51.170} C_DIS
LIN {X 0.018,Y -543.636,Z 801.081,A 0.000,B 0.000,C 90.000,E1 50.481} C_DIS
LIN {X 0.079,Y -541.118,Z 801.077,A 0.000,B 0.000,C 90.000,E1 49.908} C_DIS
LIN {X 0.067,Y -536.712,Z 801.073,A 0.000,B 0.000,C 90.000,E1 49.057} C_DIS
LIN {X -0.107,Y -534.444,Z 801.070,A 0.000,B 0.000,C 90.000,E1 48.647} C_DIS
LIN {X 0.067,Y -530.068,Z 801.066,A 0.000,B 0.000,C 90.000,E1 47.919} C_DIS
LIN {X 0.008,Y -526.169,Z 801.063,A 0.000,B 0.000,C 90.000,E1 47.349} C_DIS
LIN {X -0.111,Y -521.832,Z 801.060,A 0.000,B 0.000,C 90.000,E1 46.782} C_DIS
LIN {X 0.007,Y -517.371,Z 801.057,A 0.000,B 0.000,C 90.000,E1 46.215} C_DIS
LIN {X 0.190,Y -512.566,Z 801.054,A 0.000,B 0.000,C 90.000,E1 45.648} C_DIS
LIN {X -0.035,Y -508.561,Z 801.051,A 0.000,B 0.000,C 90.000,E1 45.243} C_DIS
LIN {X 0.023,Y -502.894,Z 801.048,A 0.000,B 0.000,C 90.000,E1 44.676} C_DIS
LIN {X 0.053,Y -498.610,Z 801.046,A 0.000,B 0.000,C 90.000,E1 44.271} C_DIS
LIN {X 0.113,Y -491.223,Z 801.042,A 0.000,B 0.000,C 90.000,E1 43.623} C_DIS
LIN {X 0.026,Y -486.653,Z 801.040,A 0.000,B 0.000,C 90.000,E1 43.257} C_DIS
LIN {X -0.001,Y -481.953,Z 801.038,A 0.000,B 0.000,C 90.000,E1 42.894} C_DIS
LIN {X -0.055,Y -474.028,Z 801.035,A 0.000,B 0.000,C 90.000,E1 42.324} C_DIS
LIN {X 0.058,Y -464.436,Z 801.031,A 0.000,B 0.000,C 90.000,E1 41.634} C_DIS
LIN {X -0.037,Y -446.865,Z 801.025,A 0.000,B 0.000,C 90.000,E1 40.415} C_DIS
LIN {X 0.013,Y -424.788,Z 801.016,A 0.000,B 0.000,C 90.000,E1 38.785} C_DIS
LIN {X -0.064,Y -409.240,Z 801.008,A 0.000,B 0.000,C 90.000,E1 37.523} C_DIS
LIN {X -0.155,Y -405.122,Z 801.006,A 0.000,B 0.000,C 90.000,E1 37.156} C_DIS
LIN {X 0.116,Y -402.264,Z 801.005,A 0.000,B 0.000,C 90.000,E1 36.790} C_DIS
LIN {X 0.080,Y -402.219,Z 801.005,A 0.000,B 0.000,C 90.000,E1 36.790} C_DIS
LIN {X -0.130,Y -394.655,Z 800.980,A 0.000,B 0.000,C 90.000,E1 32.467} C_DIS
LIN {X 0.076,Y -394.484,Z 800.979,A 0.000,B 0.000,C 90.000,E1 32.260} C_DIS
LIN {X 0.106,Y -395.785,Z 800.961,A 0.000,B 0.000,C 90.000,E1 28.899} C_DIS
LIN {X 0.059,Y -397.149,Z 800.947,A 0.000,B 0.000,C 90.000,E1 26.437} C_DIS
LIN {X 0.221,Y -398.722,Z 800.933,A 0.000,B 0.000,C 90.000,E1 23.951} C_DIS
LIN {X -0.128,Y -401.122,Z 800.916,A 0.000,B 0.000,C 90.000,E1 20.844} C_DIS
LIN {X 0.036,Y -404.752,Z 800.896,A 0.000,B 0.000,C 90.000,E1 17.330} C_DIS
LIN {X -0.227,Y -408.977,Z 800.879,A 0.000,B 0.000,C 90.000,E1 14.245} C_DIS
LIN {X -0.156,Y -413.429,Z 800.864,A 0.000,B 0.000,C 90.000,E1 11.478} C_DIS
LIN {X 0.237,Y -417.573,Z 800.850,A 0.000,B 0.000,C 90.000,E1 9.029} C_DIS
LIN {X 0.063,Y -420.657,Z 800.841,A 0.000,B 0.000,C 90.000,E1 7.352} C_DIS
LIN {X 0.091,Y -425.597,Z 800.826,A 0.000,B 0.000,C 90.000,E1 4.645} C_DIS
LIN {X 0.188,Y -430.679,Z 800.811,A 0.000,B 0.000,C 90.000,E1 1.949} C_DIS
LIN {X -0.176,Y -435.857,Z 800.797,A 0.000,B 0.000,C 90.000,E1 359.484} C_DIS
LIN {X 0.125,Y -441.005,Z 800.784,A 0.000,B 0.000,C 90.000,E1 357.135} C_DIS
LIN {X 0.179,Y -446.458,Z 800.771,A 0.000,B 0.000,C 90.000,E1 354.837} C_DIS
LIN {X -0.164,Y -451.260,Z 800.761,A 0.000,B 0.000,C 90.000,E1 352.932} C_DIS
LIN {X -0.099,Y -455.134,Z 800.752,A 0.000,B 0.000,C 90.000,E1 351.310} C_DIS
LIN {X -0.192,Y -458.336,Z 800.745,A 0.000,B 0.000,C 90.000,E1 350.038} C_DIS
LIN {X 0.052,Y -461.341,Z 800.739,A 0.000,B 0.000,C 90.000,E1 349.050} C_DIS
LIN {X -0.162,Y -462.587,Z 800.737,A 0.000,B 0.000,C 90.000,E1 348.757} C_DIS
LIN {X -0.015,Y -464.507,Z 800.735,A 0.000,B 0.000,C 90.000,E1 348.342} C_DIS
LIN {X 0.240,Y -466.520,Z 800.734,A 0.000,B 0.000,C 90.000,E1 347.993} C_DIS
LIN {X -0.174,Y -472.093,Z 800.730,A 0.000,B 0.000,C 90.000,E1 347.409} C_DIS
LIN {X -0.036,Y -480.102,Z 800.726,A 0.000,B 0.000,C 90.000,E1 346.700} C_DIS
LIN {X -0.135,Y -489.137,Z 800.722,A 0.000,B 0.000,C 90.000,E1 346.047} C_DIS
LIN {X -0.228,Y -498.639,Z 800.719,A 0.000,B 0.000,C 90.000,E1 345.408} C_DIS
LIN {X -0.148,Y -514.285,Z 800.713,A 0.000,B 0.000,C 90.000,E1 344.338} C_DIS
LIN {X -0.127,Y -526.662,Z 800.708,A 0.000,B 0.000,C 90.000,E1 343.504} C_DIS
LIN {X -0.039,Y -535.820,Z 800.705,A 0.000,B 0.000,C 90.000,E1 342.851} C_DIS
LIN {X 0.085,Y -544.895,Z 800.701,A 0.000,B 0.000,C 90.000,E1 342.181} C_DIS
LIN {X -0.054,Y -552.323,Z 800.698,A 0.000,B 0.000,C 90.000,E1 341.638} C_DIS
LIN {X 0.006,Y -560.672,Z 800.694,A 0.000,B 0.000,C 90.000,E1 340.913} C_DIS
LIN {X -0.039,Y -564.697,Z 800.692,A 0.000,B 0.000,C 90.000,E1 340.550} C_DIS
LIN {X -0.271,Y -569.896,Z 800.689,A 0.000,B 0.000,C 90.000,E1 340.061} C_DIS
LIN {X -0.206,Y -574.742,Z 800.686,A 0.000,B 0.000,C 90.000,E1 339.518} C_DIS
LIN {X -0.006,Y -579.187,Z 800.683,A 0.000,B 0.000,C 90.000,E1 338.954} C_DIS
LIN {X 0.020,Y -583.363,Z 800.680,A 0.000,B 0.000,C 90.000,E1 338.411} C_DIS
LIN {X -0.056,Y -589.204,Z 800.676,A 0.000,B 0.000,C 90.000,E1 337.614} C_DIS
LIN {X 0.155,Y -594.642,Z 800.671,A 0.000,B 0.000,C 90.000,E1 336.794} C_DIS
LIN {X 0.073,Y -602.323,Z 800.665,A 0.000,B 0.000,C 90.000,E1 335.613} C_DIS
LIN {X -0.170,Y -608.736,Z 800.659,A 0.000,B 0.000,C 90.000,E1 334.588} C_DIS
LIN {X 0.242,Y -614.097,Z 800.654,A 0.000,B 0.000,C 90.000,E1 333.640} C_DIS
LIN {X 0.160,Y -619.836,Z 800.648,A 0.000,B 0.000,C 90.000,E1 332.615} C_DIS
LIN {X 0.147,Y -624.658,Z 800.643,A 0.000,B 0.000,C 90.000,E1 331.719} C_DIS
LIN {X -0.042,Y -630.401,Z 800.637,A 0.000,B 0.000,C 90.000,E1 330.589} C_DIS
LIN {X 0.357,Y -634.277,Z 800.632,A 0.000,B 0.000,C 90.000,E1 329.793} C_DIS
LIN {X -0.038,Y -638.984,Z 800.627,A 0.000,B 0.000,C 90.000,E1 328.820} C_DIS
LIN {X -0.109,Y -642.275,Z 800.623,A 0.000,B 0.000,C 90.000,E1 328.074} C_DIS
LIN {X -0.216,Y -647.444,Z 800.616,A 0.000,B 0.000,C 90.000,E1 326.834} C_DIS
LIN {X -0.200,Y -650.392,Z 800.612,A 0.000,B 0.000,C 90.000,E1 326.087} C_DIS
LIN {X 0.200,Y -654.876,Z 800.605,A 0.000,B 0.000,C 90.000,E1 324.815} C_DIS
LIN {X 0.215,Y -658.109,Z 800.599,A 0.000,B 0.000,C 90.000,E1 323.829} C_DIS
LIN {X 0.269,Y -661.182,Z 800.594,A 0.000,B 0.000,C 90.000,E1 322.844} C_DIS
LIN {X -0.170,Y -664.133,Z 800.588,A 0.000,B 0.000,C 90.000,E1 321.904} C_DIS
LIN {X -0.080,Y -667.458,Z 800.582,A 0.000,B 0.000,C 90.000,E1 320.678} C_DIS
LIN {X -0.027,Y -670.438,Z 800.575,A 0.000,B 0.000,C 90.000,E1 319.461} C_DIS
LIN {X 0.096,Y -673.734,Z 800.567,A 0.000,B 0.000,C 90.000,E1 318.000} C_DIS
LIN {X -0.317,Y -674.817,Z 800.564,A 0.000,B 0.000,C 90.000,E1 317.553} C_DIS
LIN {X 0.313,Y -677.122,Z 800.557,A 0.000,B 0.000,C 90.000,E1 316.296} C_DIS
LIN {X -0.021,Y -678.782,Z 800.552,A 0.000,B 0.000,C 90.000,E1 315.364} C_DIS
LIN {X -0.338,Y -680.291,Z 800.547,A 0.000,B 0.000,C 90.000,E1 314.433} C_DIS
LIN {X -0.015,Y -682.634,Z 800.537,A 0.000,B 0.000,C 90.000,E1 312.732} C_DIS
LIN {X 0.230,Y -683.872,Z 800.532,A 0.000,B 0.000,C 90.000,E1 311.757} C_DIS
LIN {X -0.413,Y -685.351,Z 800.526,A 0.000,B 0.000,C 90.000,E1 310.620} C_DIS
LIN {X -0.070,Y -686.619,Z 800.519,A 0.000,B 0.000,C 90.000,E1 309.402} C_DIS
LIN {X -0.151,Y -687.787,Z 800.512,A 0.000,B 0.000,C 90.000,E1 308.222} C_DIS
LIN {X -0.043,Y -689.113,Z 800.504,A 0.000,B 0.000,C 90.000,E1 306.790} C_DIS
LIN {X 0.052,Y -690.123,Z 800.498,A 0.000,B 0.000,C 90.000,E1 305.598} C_DIS
LIN {X -0.192,Y -691.230,Z 800.490,A 0.000,B 0.000,C 90.000,E1 304.199} C_DIS
LIN {X -0.202,Y -692.440,Z 800.481,A 0.000,B 0.000,C 90.000,E1 302.546} C_DIS
LIN {X 0.030,Y -693.668,Z 800.472,A 0.000,B 0.000,C 90.000,E1 300.875} C_DIS
LIN {X 0.154,Y -694.357,Z 800.466,A 0.000,B 0.000,C 90.000,E1 299.922} C_DIS
LIN {X -0.180,Y -695.211,Z 800.458,A 0.000,B 0.000,C 90.000,E1 298.537} C_DIS
LIN {X 0.043,Y -696.185,Z 800.449,A 0.000,B 0.000,C 90.000,E1 296.873} C_DIS
LIN {X -0.371,Y -697.536,Z 800.439,A 0.000,B 0.000,C 90.000,E1 295.027} C_DIS
LIN {X 0.150,Y -697.773,Z 800.436,A 0.000,B 0.000,C 90.000,E1 294.515} C_DIS
LIN {X 0.123,Y -697.845,Z 800.435,A 0.000,B 0.000,C 90.000,E1 294.283} C_DIS
LIN {X 0.009,Y -697.454,Z 800.432,A 0.000,B 0.000,C 90.000,E1 293.823} C_DIS
LIN {X -0.012,Y -697.188,Z 800.431,A 0.000,B 0.000,C 90.000,E1 293.590} C_DIS
LIN {X 0.246,Y -696.342,Z 800.430,A 0.000,B 0.000,C 90.000,E1 293.334} C_DIS
LIN {X -0.159,Y -693.856,Z 800.427,A 0.000,B 0.000,C 90.000,E1 292.898} C_DIS
LIN {X -0.035,Y -692.938,Z 800.427,A 0.000,B 0.000,C 90.000,E1 292.770} C_DIS
LIN {X 0.087,Y -691.570,Z 800.426,A 0.000,B 0.000,C 90.000,E1 292.642} C_DIS
LIN {X 0.300,Y -689.924,Z 800.425,A 0.000,B 0.000,C 90.000,E1 292.514} C_DIS
LIN {X -0.066,Y -684.911,Z 800.424,A 0.000,B 0.000,C 90.000,E1 292.259} C_DIS
LIN {X 0.174,Y -682.976,Z 800.423,A 0.000,B 0.000,C 90.000,E1 292.153} C_DIS
LIN {X 0.241,Y -674.820,Z 800.422,A 0.000,B 0.000,C 90.000,E1 291.897} C_DIS
LIN {X 0.257,Y -672.958,Z 800.422,A 0.000,B 0.000,C 90.000,E1 291.844} C_DIS
LIN {X 0.168,Y -661.674,Z 800.420,A 0.000,B 0.000,C 90.000,E1 291.663} C_DIS
LIN {X 0.038,Y -642.311,Z 800.419,A 0.000,B 0.000,C 90.000,E1 291.354} C_DIS
LIN {X 0.154,Y -632.000,Z 800.418,A 0.000,B 0.000,C 90.000,E1 291.153} C_DIS
LIN {X 0.132,Y -618.235,Z 800.416,A 0.000,B 0.000,C 90.000,E1 290.865} C_DIS
LIN {X -0.174,Y -605.000,Z 800.414,A 0.000,B 0.000,C 90.000,E1 290.556} C_DIS
LIN {X 0.119,Y -591.947,Z 800.412,A 0.000,B 0.000,C 90.000,E1 290.120} C_DIS
LIN {X -0.291,Y -585.606,Z 800.411,A 0.000,B 0.000,C 90.000,E1 289.939} C_DIS
LIN {X 0.030,Y -576.214,Z 800.409,A 0.000,B 0.000,C 90.000,E1 289.523} C_DIS
LIN {X 0.099,Y -570.757,Z 800.407,A 0.000,B 0.000,C 90.000,E1 289.214} C_DIS
LIN {X 0.041,Y -570.696,Z 800.407,A 0.000,B 0.000,C 90.000,E1 289.214} C_DIS
LIN {X 0.045,Y -568.557,Z 800.405,A 0.000,B 0.000,C 90.000,E1 288.960} C_DIS
LIN {X -0.094,Y -568.193,Z 800.405,A 0.000,B 0.000,C 90.000,E1 288.906} C_DIS
LIN {X 0.104,Y -567.041,Z 800.403,A 0.000,B 0.000,C 90.000,E1 288.544} C_DIS
LIN {X -0.036,Y -566.993,Z 800.403,A 0.000,B 0.000,C 90.000,E1 288.489} C_DIS
LIN {X -0.098,Y -567.309,Z 800.402,A 0.000,B 0.000,C 90.000,E1 288.290} C_DIS
LIN {X 0.056,Y -567.531,Z 800.400,A 0.000,B 0.000,C 90.000,E1 288.000} C_DIS
LIN {X -0.048,Y -567.820,Z 800.399,A 0.000,B 0.000,C 90.000,E1 287.873} C_DIS
LIN {X -0.326,Y -568.268,Z 800.399,A 0.000,B 0.000,C 90.000,E1 287.764} C_DIS
LIN {X -0.086,Y -571.339,Z 800.396,A 0.000,B 0.000,C 90.000,E1 287.221} C_DIS
LIN {X -0.209,Y -575.825,Z 800.392,A 0.000,B 0.000,C 90.000,E1 286.551} C_DIS
LIN {X 0.081,Y -576.603,Z 800.391,A 0.000,B 0.000,C 90.000,E1 286.386} C_DIS
LIN {X -0.255,Y -580.263,Z 800.387,A 0.000,B 0.000,C 90.000,E1 285.607} C_DIS
LIN {X -0.229,Y -582.330,Z 800.384,A 0.000,B 0.000,C 90.000,E1 285.064} C_DIS
LIN {X 0.227,Y -583.843,Z 800.381,A 0.000,B 0.000,C 90.000,E1 284.481} C_DIS
LIN {X -0.105,Y -584.402,Z 800.379,A 0.000,B 0.000,C 90.000,E1 284.245} C_DIS
LIN {X -0.055,Y -585.215,Z 800.376,A 0.000,B 0.000,C 90.000,E1 283.703} C_DIS
LIN {X -0.140,Y -585.174,Z 800.373,A 0.000,B 0.000,C 90.000,E1 283.175} C_DIS
LIN {X -0.223,Y -584.684,Z 800.370,A 0.000,B 0.000,C 90.000,E1 282.647} C_DIS
LIN {X 0.020,Y -584.310,Z 800.369,A 0.000,B 0.000,C 90.000,E1 282.355} C_DIS
LIN {X -0.067,Y -582.648,Z 800.366,A 0.000,B 0.000,C 90.000,E1 281.827} C_DIS
LIN {X -0.167,Y -580.080,Z 800.363,A 0.000,B 0.000,C 90.000,E1 281.299} C_DIS
LIN {X 0.176,Y -579.312,Z 800.362,A 0.000,B 0.000,C 90.000,E1 281.130} C_DIS
LIN {X -0.166,Y -577.233,Z 800.360,A 0.000,B 0.000,C 90.000,E1 280.894} C_DIS
LIN {X 0.052,Y -574.870,Z 800.359,A 0.000,B 0.000,C 90.000,E1 280.602} C_DIS
LIN {X 0.026,Y -571.337,Z 800.358,A 0.000,B 0.000,C 90.000,E1 280.366} C_DIS
LIN {X 0.123,Y -568.806,Z 800.357,A 0.000,B 0.000,C 90.000,E1 280.254} C_DIS
LIN {X -0.090,Y -563.246,Z 800.356,A 0.000,B 0.000,C 90.000,E1 280.074} C_DIS
LIN {X -0.145,Y -557.735,Z 800.355,A 0.000,B 0.000,C 90.000,E1 279.905} C_DIS
LIN {X -0.083,Y -553.558,Z 800.353,A 0.000,B 0.000,C 90.000,E1 279.613} C_DIS
LIN {X -0.056,Y -552.037,Z 800.353,A 0.000,B 0.000,C 90.000,E1 279.500} C_DIS
LIN {X 0.157,Y -551.795,Z 800.353,A 0.000,B 0.000,C 90.000,E1 279.443} C_DIS
LIN {X 0.124,Y -551.792,Z 800.353,A 0.000,B 0.000,C 90.000,E1 279.443} C_DIS
LIN {X -0.227,Y -551.094,Z 800.348,A 0.000,B 0.000,C 90.000,E1 278.568} C_DIS
LIN {X 0.134,Y -550.800,Z 800.341,A 0.000,B 0.000,C 90.000,E1 277.409} C_DIS
LIN {X 0.059,Y -549.965,Z 800.330,A 0.000,B 0.000,C 90.000,E1 275.454} C_DIS
LIN {X -0.255,Y -549.532,Z 800.326,A 0.000,B 0.000,C 90.000,E1 274.645} C_DIS
LIN {X -0.029,Y -548.868,Z 800.319,A 0.000,B 0.000,C 90.000,E1 273.498} C_DIS
LIN {X -0.240,Y -547.705,Z 800.310,A 0.000,B 0.000,C 90.000,E1 271.833} C_DIS
LIN {X 0.078,Y -546.442,Z 800.299,A 0.000,B 0.000,C 90.000,E1 269.828} C_DIS
LIN {X -0.259,Y -545.417,Z 800.291,A 0.000,B 0.000,C 90.000,E1 268.453} C_DIS
LIN {X 0.063,Y -543.940,Z 800.279,A 0.000,B 0.000,C 90.000,E1 266.159} C_DIS
LIN {X -0.201,Y -542.864,Z 800.269,A 0.000,B 0.000,C 90.000,E1 264.489} C_DIS
LIN {X -0.016,Y -541.866,Z 800.261,A 0.000,B 0.000,C 90.000,E1 263.053} C_DIS
LIN {X 0.278,Y -540.691,Z 800.254,A 0.000,B 0.000,C 90.000,E1 261.602} C_DIS
LIN {X 0.028,Y -539.448,Z 800.246,A 0.000,B 0.000,C 90.000,E1 260.208} C_DIS
LIN {X -0.117,Y -537.509,Z 800.235,A 0.000,B 0.000,C 90.000,E1 258.229} C_DIS
LIN {X -0.151,Y -535.849,Z 800.225,A 0.000,B 0.000,C 90.000,E1 256.520} C_DIS
LIN {X 0.063,Y -534.593,Z 800.219,A 0.000,B 0.000,C 90.000,E1 255.353} C_DIS
LIN {X 0.011,Y -533.292,Z 800.212,A 0.000,B 0.000,C 90.000,E1 254.212} C_DIS
LIN {X 0.012,Y -531.308,Z 800.203,A 0.000,B 0.000,C 90.000,E1 252.489} C_DIS
LIN {X 0.086,Y -529.898,Z 800.196,A 0.000,B 0.000,C 90.000,E1 251.329} C_DIS
LIN {X -0.163,Y -527.664,Z 800.187,A 0.000,B 0.000,C 90.000,E1 249.625} C_DIS
LIN {X 0.041,Y -525.556,Z 800.179,A 0.000,B 0.000,C 90.000,E1 248.156} C_DIS
LIN {X -0.290,Y -523.426,Z 800.171,A 0.000,B 0.000,C 90.000,E1 246.741} C_DIS
LIN {X 0.230,Y -521.237,Z 800.163,A 0.000,B 0.000,C 90.000,E1 245.229} C_DIS
LIN {X 0.098,Y -519.364,Z 800.156,A 0.000,B 0.000,C 90.000,E1 244.076} C_DIS
LIN {X 0.071,Y -516.877,Z 800.148,A 0.000,B 0.000,C 90.000,E1 242.615} C_DIS
LIN {X 0.118,Y -514.859,Z 800.141,A 0.000,B 0.000,C 90.000,E1 241.435} C_DIS
LIN {X -0.213,Y -512.115,Z 800.133,A 0.000,B 0.000,C 90.000,E1 239.999} C_DIS
LIN {X 0.021,Y -509.809,Z 800.127,A 0.000,B 0.000,C 90.000,E1 238.791} C_DIS
LIN {X -0.257,Y -506.179,Z 800.117,A 0.000,B 0.000,C 90.000,E1 237.041} C_DIS
LIN {X -0.151,Y -504.270,Z 800.112,A 0.000,B 0.000,C 90.000,E1 236.135} C_DIS
LIN {X 0.003,Y -500.263,Z 800.102,A 0.000,B 0.000,C 90.000,E1 234.322} C_DIS
LIN {X -0.216,Y -496.507,Z 800.094,A 0.000,B 0.000,C 90.000,E1 232.844} C_DIS
LIN {X -0.050,Y -491.947,Z 800.083,A 0.000,B 0.000,C 90.000,E1 231.009} C_DIS
LIN {X 0.128,Y -485.529,Z 800.068,A 0.000,B 0.000,C 90.000,E1 228.243} C_DIS
LIN {X -0.245,Y -480.870,Z 800.056,A 0.000,B 0.000,C 90.000,E1 226.134} C_DIS
LIN {X 0.257,Y -478.132,Z 800.049,A 0.000,B 0.000,C 90.000,E1 224.838} C_DIS
LIN {X 0.144,Y -474.766,Z 800.041,A 0.000,B 0.000,C 90.000,E1 223.299} C_DIS
LIN {X -0.157,Y -470.015,Z 800.029,A 0.000,B 0.000,C 90.000,E1 221.148} C_DIS
LIN {X -0.106,Y -464.799,Z 800.015,A 0.000,B 0.000,C 90.000,E1 218.624} C_DIS
LIN {X -0.141,Y -459.500,Z 800.000,A 0.000,B 0.000,C 90.000,E1 216.091} C_DIS
LIN {X 0.296,Y -455.498,Z 799.990,A 0.000,B 0.000,C 90.000,E1 214.119} C_DIS
LIN {X -0.165,Y -450.924,Z 799.977,A 0.000,B 0.000,C 90.000,E1 211.926} C_DIS
LIN {X 0.247,Y -447.703,Z 799.968,A 0.000,B 0.000,C 90.000,E1 210.256} C_DIS
LIN {X -0.232,Y -444.476,Z 799.959,A 0.000,B 0.000,C 90.000,E1 208.693} C_DIS
LIN {X 0.066,Y -440.815,Z 799.948,A 0.000,B 0.000,C 90.000,E1 206.693} C_DIS
LIN {X 0.096,Y -436.390,Z 799.936,A 0.000,B 0.000,C 90.000,E1 204.387} C_DIS
LIN {X -0.008,Y -433.798,Z 799.928,A 0.000,B 0.000,C 90.000,E1 203.078} C_DIS
LIN {X -0.121,Y -429.966,Z 799.917,A 0.000,B 0.000,C 90.000,E1 201.099} C_DIS
LIN {X -0.084,Y -424.825,Z 799.902,A 0.000,B 0.000,C 90.000,E1 198.417} C_DIS
LIN {X -0.026,Y -420.934,Z 799.891,A 0.000,B 0.000,C 90.000,E1 196.386} C_DIS
LIN {X -0.216,Y -417.602,Z 799.882,A 0.000,B 0.000,C 90.000,E1 194.717} C_DIS
LIN {X 0.004,Y -413.135,Z 799.868,A 0.000,B 0.000,C 90.000,E1 192.299} C_DIS
LIN {X -0.057,Y -408.217,Z 799.853,A 0.000,B 0.000,C 90.000,E1 189.557} C_DIS
LIN {X 0.028,Y -405.118,Z 799.844,A 0.000,B 0.000,C 90.000,E1 187.814} C_DIS
LIN {X -0.063,Y -401.292,Z 799.832,A 0.000,B 0.000,C 90.000,E1 185.739} C_DIS
LIN {X 0.113,Y -394.206,Z 799.807,A 0.000,B 0.000,C 90.000,E1 181.146} C_DIS
LIN {X -0.003,Y -391.272,Z 799.793,A 0.000,B 0.000,C 90.000,E1 178.682} C_DIS
LIN {X -0.020,Y -389.391,Z 799.783,A 0.000,B 0.000,C 90.000,E1 176.906} C_DIS
LIN {X 0.189,Y -386.733,Z 799.769,A 0.000,B 0.000,C 90.000,E1 174.375} C_DIS
LIN {X 0.130,Y -384.850,Z 799.759,A 0.000,B 0.000,C 90.000,E1 172.591} C_DIS
LIN {X -0.168,Y -383.512,Z 799.751,A 0.000,B 0.000,C 90.000,E1 171.197} C_DIS
LIN {X 0.002,Y -380.992,Z 799.735,A 0.000,B 0.000,C 90.000,E1 168.285} C_DIS
LIN {X 0.212,Y -378.421,Z 799.715,A 0.000,B 0.000,C 90.000,E1 164.629} C_DIS
LIN {X -0.045,Y -376.386,Z 799.687,A 0.000,B 0.000,C 90.000,E1 159.571} C_DIS
LIN {X 0.009,Y -377.587,Z 799.650,A 0.000,B 0.000,C 90.000,E1 152.999} C_DIS
LIN {X 0.156,Y -379.538,Z 799.638,A 0.000,B 0.000,C 90.000,E1 150.795} C_DIS
LIN {X -0.086,Y -381.000,Z 799.632,A 0.000,B 0.000,C 90.000,E1 149.744} C_DIS
LIN {X -0.118,Y -382.977,Z 799.626,A 0.000,B 0.000,C 90.000,E1 148.663} C_DIS
LIN {X -0.122,Y -385.521,Z 799.620,A 0.000,B 0.000,C 90.000,E1 147.582} C_DIS
LIN {X 0.070,Y -387.553,Z 799.616,A 0.000,B 0.000,C 90.000,E1 146.834} C_DIS
LIN {X -0.096,Y -388.789,Z 799.614,A 0.000,B 0.000,C 90.000,E1 146.501} C_DIS
LIN {X -0.041,Y -389.869,Z 799.612,A 0.000,B 0.000,C 90.000,E1 146.135} C_DIS
LIN {X 0.190,Y -392.551,Z 799.608,A 0.000,B 0.000,C 90.000,E1 145.388} C_DIS
LIN {X 0.122,Y -395.687,Z 799.604,A 0.000,B 0.000,C 90.000,E1 144.689} C_DIS
LIN {X 0.078,Y -399.448,Z 799.600,A 0.000,B 0.000,C 90.000,E1 143.989} C_DIS
LIN {X 0.036,Y -403.246,Z 799.597,A 0.000,B 0.000,C 90.000,E1 143.371} C_DIS
LIN {X 0.214,Y -408.608,Z 799.592,A 0.000,B 0.000,C 90.000,E1 142.557} C_DIS
LIN {X 0.249,Y -416.444,Z 799.587,A 0.000,B 0.000,C 90.000,E1 141.537} C_DIS
LIN {X 0.101,Y -424.760,Z 799.581,A 0.000,B 0.000,C 90.000,E1 140.561} C_DIS
LIN {X -0.102,Y -432.546,Z 799.575,A 0.000,B 0.000,C 90.000,E1 139.585} C_DIS
LIN {X -0.012,Y -446.603,Z 799.565,A 0.000,B 0.000,C 90.000,E1 137.757} C_DIS
LIN {X -0.131,Y -454.206,Z 799.560,A 0.000,B 0.000,C 90.000,E1 136.824} C_DIS
LIN {X -0.095,Y -461.266,Z 799.555,A 0.000,B 0.000,C 90.000,E1 135.891} C_DIS
LIN {X 0.009,Y -464.750,Z 799.552,A 0.000,B 0.000,C 90.000,E1 135.405} C_DIS
LIN {X -0.038,Y -475.509,Z 799.544,A 0.000,B 0.000,C 90.000,E1 133.866} C_DIS
LIN {X -0.040,Y -481.859,Z 799.539,A 0.000,B 0.000,C 90.000,E1 132.933} C_DIS
LIN {X 0.033,Y -487.840,Z 799.533,A 0.000,B 0.000,C 90.000,E1 132.000} C_DIS
LIN {X 0.090,Y -495.397,Z 799.527,A 0.000,B 0.000,C 90.000,E1 130.782} C_DIS
LIN {X 0.212,Y -502.411,Z 799.520,A 0.000,B 0.000,C 90.000,E1 129.564} C_DIS
LIN {X 0.194,Y -507.506,Z 799.515,A 0.000,B 0.000,C 90.000,E1 128.669} C_DIS
LIN {X -0.175,Y -513.819,Z 799.508,A 0.000,B 0.000,C 90.000,E1 127.523} C_DIS
LIN {X -0.206,Y -517.556,Z 799.504,A 0.000,B 0.000,C 90.000,E1 126.790} C_DIS
LIN {X -0.013,Y -523.276,Z 799.498,A 0.000,B 0.000,C 90.000,E1 125.598} C_DIS
LIN {X -0.133,Y -527.207,Z 799.493,A 0.000,B 0.000,C 90.000,E1 124.739} C_DIS
LIN {X -0.115,Y -533.175,Z 799.485,A 0.000,B 0.000,C 90.000,E1 123.293} C_DIS
LIN {X 0.010,Y -536.585,Z 799.480,A 0.000,B 0.000,C 90.000,E1 122.418} C_DIS
LIN {X 0.179,Y -540.838,Z 799.474,A 0.000,B 0.000,C 90.000,E1 121.258} C_DIS
LIN {X 0.114,Y -543.840,Z 799.469,A 0.000,B 0.000,C 90.000,E1 120.413} C_DIS
LIN {X 0.108,Y -547.510,Z 799.463,A 0.000,B 0.000,C 90.000,E1 119.283} C_DIS
LIN {X 0.145,Y -550.867,Z 799.457,A 0.000,B 0.000,C 90.000,E1 118.153} C_DIS
LIN {X -0.064,Y -553.196,Z 799.452,A 0.000,B 0.000,C 90.000,E1 117.334} C_DIS
LIN {X 0.009,Y -555.184,Z 799.447,A 0.000,B 0.000,C 90.000,E1 116.488} C_DIS
LIN {X -0.121,Y -557.216,Z 799.441,A 0.000,B 0.000,C 90.000,E1 115.387} C_DIS
LIN {X -0.046,Y -558.185,Z 799.438,A 0.000,B 0.000,C 90.000,E1 114.823} C_DIS
LIN {X 0.130,Y -559.568,Z 799.432,A 0.000,B 0.000,C 90.000,E1 113.695} C_DIS
LIN {X -0.100,Y -561.071,Z 799.424,A 0.000,B 0.000,C 90.000,E1 112.333} C_DIS
LIN {X -0.095,Y -562.186,Z 799.418,A 0.000,B 0.000,C 90.000,E1 111.227} C_DIS
LIN {X 0.244,Y -563.261,Z 799.410,A 0.000,B 0.000,C 90.000,E1 109.812} C_DIS
LIN {X -0.129,Y -563.944,Z 799.403,A 0.000,B 0.000,C 90.000,E1 108.471} C_DIS
LIN {X -0.135,Y -564.569,Z 799.395,A 0.000,B 0.000,C 90.000,E1 107.094} C_DIS
LIN {X 0.032,Y -565.407,Z 799.386,A 0.000,B 0.000,C 90.000,E1 105.426} C_DIS
LIN {X -0.133,Y -566.795,Z 799.374,A 0.000,B 0.000,C 90.000,E1 103.244} C_DIS
LIN {X -0.069,Y -567.951,Z 799.364,A 0.000,B 0.000,C 90.000,E1 101.591} C_DIS
LIN {X -0.034,Y -569.414,Z 799.354,A 0.000,B 0.000,C 90.000,E1 99.670} C_DIS
LIN {X 0.044,Y -570.257,Z 799.348,A 0.000,B 0.000,C 90.000,E1 98.568} C_DIS
LIN {X 0.239,Y -571.205,Z 799.340,A 0.000,B 0.000,C 90.000,E1 97.182} C_DIS
LIN {X -0.116,Y -572.039,Z 799.333,A 0.000,B 0.000,C 90.000,E1 95.853} C_DIS
LIN {X 0.183,Y -572.952,Z 799.323,A 0.000,B 0.000,C 90.000,E1 94.188} C_DIS
LIN {X -0.068,Y -573.698,Z 799.314,A 0.000,B 0.000,C 90.000,E1 92.579} C_DIS
LIN {X 0.092,Y -574.278,Z 799.307,A 0.000,B 0.000,C 90.000,E1 91.203} C_DIS
LIN {X -0.030,Y -574.895,Z 799.296,A 0.000,B 0.000,C 90.000,E1 89.312} C_DIS
LIN {X 0.153,Y -575.332,Z 799.289,A 0.000,B 0.000,C 90.000,E1 87.936} C_DIS
LIN {X -0.228,Y -575.690,Z 799.281,A 0.000,B 0.000,C 90.000,E1 86.617} C_DIS
LIN {X -0.280,Y -576.150,Z 799.271,A 0.000,B 0.000,C 90.000,E1 84.723} C_DIS
LIN {X 0.151,Y -576.436,Z 799.262,A 0.000,B 0.000,C 90.000,E1 83.053} C_DIS
LIN {X -0.121,Y -576.703,Z 799.254,A 0.000,B 0.000,C 90.000,E1 81.724} C_DIS
LIN {X -0.089,Y -577.001,Z 799.245,A 0.000,B 0.000,C 90.000,E1 80.095} C_DIS
LIN {X 0.092,Y -577.219,Z 799.239,A 0.000,B 0.000,C 90.000,E1 78.993} C_DIS
LIN {X 0.031,Y -577.301,Z 799.231,A 0.000,B 0.000,C 90.000,E1 77.645} C_DIS
LIN {X 0.320,Y -577.244,Z 799.222,A 0.000,B 0.000,C 90.000,E1 75.992} C_DIS
LIN {X -0.155,Y -577.077,Z 799.215,A 0.000,B 0.000,C 90.000,E1 74.685} C_DIS
LIN {X 0.117,Y -576.830,Z 799.206,A 0.000,B 0.000,C 90.000,E1 73.032} C_DIS
LIN {X 0.156,Y -576.503,Z 799.197,A 0.000,B 0.000,C 90.000,E1 71.402} C_DIS
LIN {X -0.157,Y -575.944,Z 799.188,A 0.000,B 0.000,C 90.000,E1 69.806} C_DIS
LIN {X -0.145,Y -575.524,Z 799.182,A 0.000,B 0.000,C 90.000,E1 68.720} C_DIS
LIN {X 0.269,Y -574.732,Z 799.173,A 0.000,B 0.000,C 90.000,E1 67.050} C_DIS
LIN {X 0.160,Y -574.107,Z 799.167,A 0.000,B 0.000,C 90.000,E1 65.973} C_DIS
LIN {X -0.353,Y -573.248,Z 799.159,A 0.000,B 0.000,C 90.000,E1 64.665} C_DIS
LIN {X 0.286,Y -572.454,Z 799.153,A 0.000,B 0.000,C 90.000,E1 63.512} C_DIS
LIN {X 0.140,Y -571.470,Z 799.147,A 0.000,B 0.000,C 90.000,E1 62.436} C_DIS
LIN {X -0.093,Y -570.609,Z 799.142,A 0.000,B 0.000,C 90.000,E1 61.641} C_DIS
LIN {X -0.004,Y -569.280,Z 799.136,A 0.000,B 0.000,C 90.000,E1 60.539} C_DIS
LIN {X -0.147,Y -567.743,Z 799.130,A 0.000,B 0.000,C 90.000,E1 59.459} C_DIS
LIN {X 0.181,Y -565.970,Z 799.124,A 0.000,B 0.000,C 90.000,E1 58.329} C_DIS
LIN {X -0.104,Y -564.460,Z 799.120,A 0.000,B 0.000,C 90.000,E1 57.533} C_DIS
LIN {X -0.104,Y -562.783,Z 799.115,A 0.000,B 0.000,C 90.000,E1 56.707} C_DIS
LIN {X -0.120,Y -560.971,Z 799.110,A 0.000,B 0.000,C 90.000,E1 55.881} C_DIS
LIN {X -0.067,Y -558.119,Z 799.104,A 0.000,B 0.000,C 90.000,E1 54.769} C_DIS
LIN {X 0.106,Y -556.627,Z 799.101,A 0.000,B 0.000,C 90.000,E1 54.196} C_DIS
LIN {X 0.088,Y -553.177,Z 799.095,A 0.000,B 0.000,C 90.000,E1 53.084} C_DIS
LIN {X -0.151,Y -550.304,Z 799.090,A 0.000,B 0.000,C 90.000,E1 52.271} C_DIS
LIN {X -0.091,Y -549.312,Z 799.089,A 0.000,B 0.000,C 90.000,E1 51.984} C_DIS
LIN {X 0.063,Y -545.941,Z 799.084,A 0.000,B 0.000,C 90.000,E1 51.126} C_DIS
LIN {X -0.090,Y -542.867,Z 799.080,A 0.000,B 0.000,C 90.000,E1 50.436} C_DIS
LIN {X 0.310,Y -540.240,Z 799.077,A 0.000,B 0.000,C 90.000,E1 49.828} C_DIS
LIN {X 0.109,Y -536.502,Z 799.073,A 0.000,B 0.000,C 90.000,E1 49.138} C_DIS
LIN {X 0.108,Y -533.347,Z 799.070,A 0.000,B 0.000,C 90.000,E1 48.566} C_DIS
LIN {X 0.123,Y -529.798,Z 799.067,A 0.000,B 0.000,C 90.000,E1 48.000} C_DIS
LIN {X -0.325,Y -525.872,Z 799.064,A 0.000,B 0.000,C 90.000,E1 47.472} C_DIS
LIN {X -0.060,Y -521.510,Z 799.060,A 0.000,B 0.000,C 90.000,E1 46.863} C_DIS
LIN {X 0.069,Y -516.987,Z 799.057,A 0.000,B 0.000,C 90.000,E1 46.296} C_DIS
LIN {X -0.313,Y -510.746,Z 799.053,A 0.000,B 0.000,C 90.000,E1 45.648} C_DIS
LIN {X 0.020,Y -508.089,Z 799.052,A 0.000,B 0.000,C 90.000,E1 45.324} C_DIS
LIN {X 0.178,Y -502.441,Z 799.049,A 0.000,B 0.000,C 90.000,E1 44.757} C_DIS
LIN {X 0.215,Y -498.136,Z 799.047,A 0.000,B 0.000,C 90.000,E1 44.352} C_DIS
LIN {X 0.203,Y -490.594,Z 799.043,A 0.000,B 0.000,C 90.000,E1 43.704} C_DIS
LIN {X -0.046,Y -483.093,Z 799.040,A 0.000,B 0.000,C 90.000,E1 43.137} C_DIS
LIN {X 0.147,Y -475.090,Z 799.036,A 0.000,B 0.000,C 90.000,E1 42.528} C_DIS
LIN {X 0.242,Y -465.495,Z 799.033,A 0.000,B 0.000,C 90.000,E1 41.838} C_DIS
LIN {X 0.169,Y -447.846,Z 799.026,A 0.000,B 0.000,C 90.000,E1 40.620} C_DIS
LIN {X 0.151,Y -422.447,Z 799.015,A 0.000,B 0.000,C 90.000,E1 38.749} C_DIS
LIN {X 0.265,Y -410.197,Z 799.010,A 0.000,B 0.000,C 90.000,E1 37.729} C_DIS
LIN {X 0.148,Y -405.936,Z 799.008,A 0.000,B 0.000,C 90.000,E1 37.363} C_DIS
LIN {X 0.097,Y -404.656,Z 799.007,A 0.000,B 0.000,C 90.000,E1 37.237} C_DIS
LIN {X -0.028,Y -402.623,Z 799.006,A 0.000,B 0.000,C 90.000,E1 36.996} C_DIS
LIN {X -0.062,Y -402.602,Z 799.006,A 0.000,B 0.000,C 90.000,E1 36.996} C_DIS
LIN {X 0.089,Y -394.815,Z 798.981,A 0.000,B 0.000,C 90.000,E1 32.546} C_DIS
LIN {X -0.248,Y -394.705,Z 798.980,A 0.000,B 0.000,C 90.000,E1 32.418} C_DIS
LIN {X -0.033,Y -395.996,Z 798.961,A 0.000,B 0.000,C 90.000,E1 29.027} C_DIS
LIN {X 0.101,Y -397.328,Z 798.948,A 0.000,B 0.000,C 90.000,E1 26.539} C_DIS
LIN {X 0.164,Y -398.408,Z 798.938,A 0.000,B 0.000,C 90.000,E1 24.771} C_DIS
LIN {X -0.038,Y -400.710,Z 798.920,A 0.000,B 0.000,C 90.000,E1 21.642} C_DIS
LIN {X 0.112,Y -404.100,Z 798.901,A 0.000,B 0.000,C 90.000,E1 18.127} C_DIS
LIN {X 0.176,Y -409.097,Z 798.880,A 0.000,B 0.000,C 90.000,E1 14.300} C_DIS
LIN {X -0.155,Y -413.543,Z 798.864,A 0.000,B 0.000,C 90.000,E1 11.591} C_DIS
LIN {X 0.115,Y -417.052,Z 798.853,A 0.000,B 0.000,C 90.000,E1 9.500} C_DIS
LIN {X -0.005,Y -420.098,Z 798.843,A 0.000,B 0.000,C 90.000,E1 7.814} C_DIS
LIN {X -0.179,Y -423.155,Z 798.834,A 0.000,B 0.000,C 90.000,E1 6.144} C_DIS
LIN {X 0.131,Y -426.260,Z 798.825,A 0.000,B 0.000,C 90.000,E1 4.416} C_DIS
LIN {X 0.182,Y -430.744,Z 798.812,A 0.000,B 0.000,C 90.000,E1 2.064} C_DIS
LIN {X -0.175,Y -436.113,Z 798.797,A 0.000,B 0.000,C 90.000,E1 359.484} C_DIS
LIN {X 0.133,Y -441.252,Z 798.784,A 0.000,B 0.000,C 90.000,E1 357.135} C_DIS
LIN {X 0.193,Y -446.688,Z 798.771,A 0.000,B 0.000,C 90.000,E1 354.837} C_DIS
LIN {X -0.144,Y -451.459,Z 798.761,A 0.000,B 0.000,C 90.000,E1 352.932} C_DIS
LIN {X -0.075,Y -455.330,Z 798.752,A 0.000,B 0.000,C 90.000,E1 351.310} C_DIS
LIN {X 0.065,Y -459.319,Z 798.743,A 0.000,B 0.000,C 90.000,E1 349.690} C_DIS
LIN {X 0.081,Y -461.296,Z 798.739,A 0.000,B 0.000,C 90.000,E1 349.050} C_DIS
LIN {X 0.035,Y -463.076,Z 798.737,A 0.000,B 0.000,C 90.000,E1 348.578} C_DIS
LIN {X -0.094,Y -465.398,Z 798.734,A 0.000,B 0.000,C 90.000,E1 348.117} C_DIS
LIN {X 0.234,Y -467.925,Z 798.732,A 0.000,B 0.000,C 90.000,E1 347.701} C_DIS
LIN {X -0.107,Y -471.885,Z 798.729,A 0.000,B 0.000,C 90.000,E1 347.285} C_DIS
